(* IEC 61131-3 sources: elnaProjects/ElpcLogic/PomarKc7Changed/build_USO_ecl (part 2) *)

  ai.Tstali_statora_kanal_1.inCommand_ARM := UINT_TO_WORD(AI_Tstali_statora_kanal_1_command);
  ai.Tstali_statora_kanal_1.dHL := AI_Tstali_statora_kanal_1_newHL;
  ai.Tstali_statora_kanal_1.dLL := AI_Tstali_statora_kanal_1_newLL;
  ai.Tstali_statora_kanal_1.dHW := AI_Tstali_statora_kanal_1_newHW;

  ai.Tstali_statora_kanal_2.inCommand_ARM := UINT_TO_WORD(AI_Tstali_statora_kanal_2_command);
  ai.Tstali_statora_kanal_2.dHL := AI_Tstali_statora_kanal_2_newHL;
  ai.Tstali_statora_kanal_2.dLL := AI_Tstali_statora_kanal_2_newLL;
  ai.Tstali_statora_kanal_2.dHW := AI_Tstali_statora_kanal_2_newHW;

  ai.Tstali_statora_kanal_3.inCommand_ARM := UINT_TO_WORD(AI_Tstali_statora_kanal_3_command);
  ai.Tstali_statora_kanal_3.dHL := AI_Tstali_statora_kanal_3_newHL;
  ai.Tstali_statora_kanal_3.dLL := AI_Tstali_statora_kanal_3_newLL;
  ai.Tstali_statora_kanal_3.dHW := AI_Tstali_statora_kanal_3_newHW;

  ai.Tmedi_statora_kanal_1.inCommand_ARM := UINT_TO_WORD(AI_Tmedi_statora_kanal_1_command);
  ai.Tmedi_statora_kanal_1.dHL := AI_Tmedi_statora_kanal_1_newHL;
  ai.Tmedi_statora_kanal_1.dLL := AI_Tmedi_statora_kanal_1_newLL;
  ai.Tmedi_statora_kanal_1.dHW := AI_Tmedi_statora_kanal_1_newHW;

  ai.Tmedi_statora_kanal_2.inCommand_ARM := UINT_TO_WORD(AI_Tmedi_statora_kanal_2_command);
  ai.Tmedi_statora_kanal_2.dHL := AI_Tmedi_statora_kanal_2_newHL;
  ai.Tmedi_statora_kanal_2.dLL := AI_Tmedi_statora_kanal_2_newLL;
  ai.Tmedi_statora_kanal_2.dHW := AI_Tmedi_statora_kanal_2_newHW;

  ai.Tmedi_statora_kanal_3.inCommand_ARM := UINT_TO_WORD(AI_Tmedi_statora_kanal_3_command);
  ai.Tmedi_statora_kanal_3.dHL := AI_Tmedi_statora_kanal_3_newHL;
  ai.Tmedi_statora_kanal_3.dLL := AI_Tmedi_statora_kanal_3_newLL;
  ai.Tmedi_statora_kanal_3.dHW := AI_Tmedi_statora_kanal_3_newHW;

  ai.Toporno_podshipnika_EDT_1.inCommand_ARM := UINT_TO_WORD(AI_Toporno_podshipnika_EDT_1_command);
  ai.Toporno_podshipnika_EDT_1.dHL := AI_Toporno_podshipnika_EDT_1_newHL;
  ai.Toporno_podshipnika_EDT_1.dLL := AI_Toporno_podshipnika_EDT_1_newLL;
  ai.Toporno_podshipnika_EDT_1.dHW := AI_Toporno_podshipnika_EDT_1_newHW;
  ai.Toporno_podshipnika_EDT_1.dHA := AI_Toporno_podshipnika_EDT_1_newHA;

  ai.Toy_podshipnika_EDT_2.inCommand_ARM := UINT_TO_WORD(AI_Toy_podshipnika_EDT_2_command);
  ai.Toy_podshipnika_EDT_2.dHL := AI_Toy_podshipnika_EDT_2_newHL;
  ai.Toy_podshipnika_EDT_2.dLL := AI_Toy_podshipnika_EDT_2_newLL;
  ai.Toy_podshipnika_EDT_2.dHW := AI_Toy_podshipnika_EDT_2_newHW;
  ai.Toy_podshipnika_EDT_2.dHA := AI_Toy_podshipnika_EDT_2_newHA;

  ai.Toy_podshipnika_kol_EDT_3.inCommand_ARM := UINT_TO_WORD(AI_Toy_podshipnika_kol_EDT_3_command);
  ai.Toy_podshipnika_kol_EDT_3.dHL := AI_Toy_podshipnika_kol_EDT_3_newHL;
  ai.Toy_podshipnika_kol_EDT_3.dLL := AI_Toy_podshipnika_kol_EDT_3_newLL;
  ai.Toy_podshipnika_kol_EDT_3.dHW := AI_Toy_podshipnika_kol_EDT_3_newHW;
  ai.Toy_podshipnika_kol_EDT_3.dHA := AI_Toy_podshipnika_kol_EDT_3_newHA;

  ai.Toy_podshipnika_kol_EDT_4.inCommand_ARM := UINT_TO_WORD(AI_Toy_podshipnika_kol_EDT_4_command);
  ai.Toy_podshipnika_kol_EDT_4.dHL := AI_Toy_podshipnika_kol_EDT_4_newHL;
  ai.Toy_podshipnika_kol_EDT_4.dLL := AI_Toy_podshipnika_kol_EDT_4_newLL;
  ai.Toy_podshipnika_kol_EDT_4.dHW := AI_Toy_podshipnika_kol_EDT_4_newHW;
  ai.Toy_podshipnika_kol_EDT_4.dHA := AI_Toy_podshipnika_kol_EDT_4_newHA;

  ai.Toy_podshipnika_shest_red_EDT_5.inCommand_ARM := UINT_TO_WORD(AI_Toy_podshipnika_shest_red_EDT_5_command);
  ai.Toy_podshipnika_shest_red_EDT_5.dHL := AI_Toy_podshipnika_shest_red_EDT_5_newHL;
  ai.Toy_podshipnika_shest_red_EDT_5.dLL := AI_Toy_podshipnika_shest_red_EDT_5_newLL;
  ai.Toy_podshipnika_shest_red_EDT_5.dHW := AI_Toy_podshipnika_shest_red_EDT_5_newHW;
  ai.Toy_podshipnika_shest_red_EDT_5.dHA := AI_Toy_podshipnika_shest_red_EDT_5_newHA;

  ai.Ty_podshipnika_red_EDT_6.inCommand_ARM := UINT_TO_WORD(AI_Ty_podshipnika_red_EDT_6_command);
  ai.Ty_podshipnika_red_EDT_6.dHL := AI_Ty_podshipnika_red_EDT_6_newHL;
  ai.Ty_podshipnika_red_EDT_6.dLL := AI_Ty_podshipnika_red_EDT_6_newLL;
  ai.Ty_podshipnika_red_EDT_6.dHW := AI_Ty_podshipnika_red_EDT_6_newHW;
  ai.Ty_podshipnika_red_EDT_6.dHA := AI_Ty_podshipnika_red_EDT_6_newHA;

  ai.Ty_podshipnika_nagnet_EDT_7_1.inCommand_ARM := UINT_TO_WORD(AI_Ty_podshipnika_nagnet_EDT_7_1_command);
  ai.Ty_podshipnika_nagnet_EDT_7_1.dHL := AI_Ty_podshipnika_nagnet_EDT_7_1_newHL;
  ai.Ty_podshipnika_nagnet_EDT_7_1.dLL := AI_Ty_podshipnika_nagnet_EDT_7_1_newLL;
  ai.Ty_podshipnika_nagnet_EDT_7_1.dHW := AI_Ty_podshipnika_nagnet_EDT_7_1_newHW;
  ai.Ty_podshipnika_nagnet_EDT_7_1.dHA := AI_Ty_podshipnika_nagnet_EDT_7_1_newHA;

  ai.Ty_podshipnika_nagnet_EDT_7_2.inCommand_ARM := UINT_TO_WORD(AI_Ty_podshipnika_nagnet_EDT_7_2_command);
  ai.Ty_podshipnika_nagnet_EDT_7_2.dHL := AI_Ty_podshipnika_nagnet_EDT_7_2_newHL;
  ai.Ty_podshipnika_nagnet_EDT_7_2.dLL := AI_Ty_podshipnika_nagnet_EDT_7_2_newLL;
  ai.Ty_podshipnika_nagnet_EDT_7_2.dHW := AI_Ty_podshipnika_nagnet_EDT_7_2_newHW;
  ai.Ty_podshipnika_nagnet_EDT_7_2.dHA := AI_Ty_podshipnika_nagnet_EDT_7_2_newHA;

  ai.Toy_podshipnika_svobod_konca_EDT_8_1.inCommand_ARM := UINT_TO_WORD(AI_Toy_podshipnika_svobod_konca_EDT_8_1_command);
  ai.Toy_podshipnika_svobod_konca_EDT_8_1.dHL := AI_Toy_podshipnika_svobod_konca_EDT_8_1_newHL;
  ai.Toy_podshipnika_svobod_konca_EDT_8_1.dLL := AI_Toy_podshipnika_svobod_konca_EDT_8_1_newLL;
  ai.Toy_podshipnika_svobod_konca_EDT_8_1.dHW := AI_Toy_podshipnika_svobod_konca_EDT_8_1_newHW;
  ai.Toy_podshipnika_svobod_konca_EDT_8_1.dHA := AI_Toy_podshipnika_svobod_konca_EDT_8_1_newHA;

  ai.Toy_podshipnika_svobod_konca_EDT_8_2.inCommand_ARM := UINT_TO_WORD(AI_Toy_podshipnika_svobod_konca_EDT_8_2_command);
  ai.Toy_podshipnika_svobod_konca_EDT_8_2.dHL := AI_Toy_podshipnika_svobod_konca_EDT_8_2_newHL;
  ai.Toy_podshipnika_svobod_konca_EDT_8_2.dLL := AI_Toy_podshipnika_svobod_konca_EDT_8_2_newLL;
  ai.Toy_podshipnika_svobod_konca_EDT_8_2.dHW := AI_Toy_podshipnika_svobod_konca_EDT_8_2_newHW;
  ai.Toy_podshipnika_svobod_konca_EDT_8_2.dHA := AI_Toy_podshipnika_svobod_konca_EDT_8_2_newHA;

  ai.Toy_podshipnika_rab_kol_EDT_9_1.inCommand_ARM := UINT_TO_WORD(AI_Toy_podshipnika_rab_kol_EDT_9_1_command);
  ai.Toy_podshipnika_rab_kol_EDT_9_1.dHL := AI_Toy_podshipnika_rab_kol_EDT_9_1_newHL;
  ai.Toy_podshipnika_rab_kol_EDT_9_1.dLL := AI_Toy_podshipnika_rab_kol_EDT_9_1_newLL;
  ai.Toy_podshipnika_rab_kol_EDT_9_1.dHW := AI_Toy_podshipnika_rab_kol_EDT_9_1_newHW;
  ai.Toy_podshipnika_rab_kol_EDT_9_1.dHA := AI_Toy_podshipnika_rab_kol_EDT_9_1_newHA;

  ai.Toy_podshipnika_rab_kol_EDT_9_2.inCommand_ARM := UINT_TO_WORD(AI_Toy_podshipnika_rab_kol_EDT_9_2_command);
  ai.Toy_podshipnika_rab_kol_EDT_9_2.dHL := AI_Toy_podshipnika_rab_kol_EDT_9_2_newHL;
  ai.Toy_podshipnika_rab_kol_EDT_9_2.dLL := AI_Toy_podshipnika_rab_kol_EDT_9_2_newLL;
  ai.Toy_podshipnika_rab_kol_EDT_9_2.dHW := AI_Toy_podshipnika_rab_kol_EDT_9_2_newHW;
  ai.Toy_podshipnika_rab_kol_EDT_9_2.dHA := AI_Toy_podshipnika_rab_kol_EDT_9_2_newHA;

  ai.Toy_podshipnika_nerab_kol_EDT_10_1.inCommand_ARM := UINT_TO_WORD(AI_Toy_podshipnika_nerab_kol_EDT_10_1_command);
  ai.Toy_podshipnika_nerab_kol_EDT_10_1.dHL := AI_Toy_podshipnika_nerab_kol_EDT_10_1_newHL;
  ai.Toy_podshipnika_nerab_kol_EDT_10_1.dLL := AI_Toy_podshipnika_nerab_kol_EDT_10_1_newLL;
  ai.Toy_podshipnika_nerab_kol_EDT_10_1.dHW := AI_Toy_podshipnika_nerab_kol_EDT_10_1_newHW;
  ai.Toy_podshipnika_nerab_kol_EDT_10_1.dHA := AI_Toy_podshipnika_nerab_kol_EDT_10_1_newHA;

  ai.Toy_podshipnika_nerab_kol_EDT_10_2.inCommand_ARM := UINT_TO_WORD(AI_Toy_podshipnika_nerab_kol_EDT_10_2_command);
  ai.Toy_podshipnika_nerab_kol_EDT_10_2.dHL := AI_Toy_podshipnika_nerab_kol_EDT_10_2_newHL;
  ai.Toy_podshipnika_nerab_kol_EDT_10_2.dLL := AI_Toy_podshipnika_nerab_kol_EDT_10_2_newLL;
  ai.Toy_podshipnika_nerab_kol_EDT_10_2.dHW := AI_Toy_podshipnika_nerab_kol_EDT_10_2_newHW;
  ai.Toy_podshipnika_nerab_kol_EDT_10_2.dHA := AI_Toy_podshipnika_nerab_kol_EDT_10_2_newHA;

  ai.Tholodnogo_vozduha_ED_kanal_1.inCommand_ARM := UINT_TO_WORD(AI_Tholodnogo_vozduha_ED_kanal_1_command);
  ai.Tholodnogo_vozduha_ED_kanal_1.dHL := AI_Tholodnogo_vozduha_ED_kanal_1_newHL;
  ai.Tholodnogo_vozduha_ED_kanal_1.dLL := AI_Tholodnogo_vozduha_ED_kanal_1_newLL;
  ai.Tholodnogo_vozduha_ED_kanal_1.dHW := AI_Tholodnogo_vozduha_ED_kanal_1_newHW;

  ai.Tholodnogo_vozduha_ED_kanal_2.inCommand_ARM := UINT_TO_WORD(AI_Tholodnogo_vozduha_ED_kanal_2_command);
  ai.Tholodnogo_vozduha_ED_kanal_2.dHL := AI_Tholodnogo_vozduha_ED_kanal_2_newHL;
  ai.Tholodnogo_vozduha_ED_kanal_2.dLL := AI_Tholodnogo_vozduha_ED_kanal_2_newLL;
  ai.Tholodnogo_vozduha_ED_kanal_2.dHW := AI_Tholodnogo_vozduha_ED_kanal_2_newHW;

  ai.Tgorjachego_vozduha_ED_kanal_1.inCommand_ARM := UINT_TO_WORD(AI_Tgorjachego_vozduha_ED_kanal_1_command);
  ai.Tgorjachego_vozduha_ED_kanal_1.dHL := AI_Tgorjachego_vozduha_ED_kanal_1_newHL;
  ai.Tgorjachego_vozduha_ED_kanal_1.dLL := AI_Tgorjachego_vozduha_ED_kanal_1_newLL;
  ai.Tgorjachego_vozduha_ED_kanal_1.dHW := AI_Tgorjachego_vozduha_ED_kanal_1_newHW;

  ai.Tgorjachego_vozduha_ED_kanal_2.inCommand_ARM := UINT_TO_WORD(AI_Tgorjachego_vozduha_ED_kanal_2_command);
  ai.Tgorjachego_vozduha_ED_kanal_2.dHL := AI_Tgorjachego_vozduha_ED_kanal_2_newHL;
  ai.Tgorjachego_vozduha_ED_kanal_2.dLL := AI_Tgorjachego_vozduha_ED_kanal_2_newLL;
  ai.Tgorjachego_vozduha_ED_kanal_2.dHW := AI_Tgorjachego_vozduha_ED_kanal_2_newHW;

  ai.Tnarujnogo_vozduha.inCommand_ARM := UINT_TO_WORD(AI_Tnarujnogo_vozduha_command);
  ai.Tnarujnogo_vozduha.dHL := AI_Tnarujnogo_vozduha_newHL;
  ai.Tnarujnogo_vozduha.dLL := AI_Tnarujnogo_vozduha_newLL;
  ai.Tnarujnogo_vozduha.dHW := AI_Tnarujnogo_vozduha_newHW;

  ai.Tgaza_na_vhode_H.inCommand_ARM := UINT_TO_WORD(AI_Tgaza_na_vhode_H_command);
  ai.Tgaza_na_vhode_H.dHL := AI_Tgaza_na_vhode_H_newHL;
  ai.Tgaza_na_vhode_H.dLL := AI_Tgaza_na_vhode_H_newLL;
  ai.Tgaza_na_vhode_H.dHW := AI_Tgaza_na_vhode_H_newHW;

  ai.Tgaza_na_vyhode_H.inCommand_ARM := UINT_TO_WORD(AI_Tgaza_na_vyhode_H_command);
  ai.Tgaza_na_vyhode_H.dHL := AI_Tgaza_na_vyhode_H_newHL;
  ai.Tgaza_na_vyhode_H.dLL := AI_Tgaza_na_vyhode_H_newLL;
  ai.Tgaza_na_vyhode_H.dHW := AI_Tgaza_na_vyhode_H_newHW;
  ai.Tgaza_na_vyhode_H.dHA := AI_Tgaza_na_vyhode_H_newHA;

  ai.Tmasla_do_AVOM.inCommand_ARM := UINT_TO_WORD(AI_Tmasla_do_AVOM_command);
  ai.Tmasla_do_AVOM.dHL := AI_Tmasla_do_AVOM_newHL;
  ai.Tmasla_do_AVOM.dLL := AI_Tmasla_do_AVOM_newLL;
  ai.Tmasla_do_AVOM.dHW := AI_Tmasla_do_AVOM_newHW;

  ai.Tmasla_posle_AVOM.inCommand_ARM := UINT_TO_WORD(AI_Tmasla_posle_AVOM_command);
  ai.Tmasla_posle_AVOM.dHL := AI_Tmasla_posle_AVOM_newHL;
  ai.Tmasla_posle_AVOM.dLL := AI_Tmasla_posle_AVOM_newLL;
  ai.Tmasla_posle_AVOM.dHW := AI_Tmasla_posle_AVOM_newHW;

  ai.Tmasla_MB.inCommand_ARM := UINT_TO_WORD(AI_Tmasla_MB_command);
  ai.Tmasla_MB.dHL := AI_Tmasla_MB_newHL;
  ai.Tmasla_MB.dLL := AI_Tmasla_MB_newLL;
  ai.Tmasla_MB.dHW := AI_Tmasla_MB_newHW;

  ai.Tmasla_MB_TEN.inCommand_ARM := UINT_TO_WORD(AI_Tmasla_MB_TEN_command);
  ai.Tmasla_MB_TEN.dHL := AI_Tmasla_MB_TEN_newHL;
  ai.Tmasla_MB_TEN.dLL := AI_Tmasla_MB_TEN_newLL;
  ai.Tmasla_MB_TEN.dHW := AI_Tmasla_MB_TEN_newHW;

  ai.Tshu.inCommand_ARM := UINT_TO_WORD(AI_Tshu_command);
  ai.Tshu.dHL := AI_Tshu_newHL;
  ai.Tshu.dLL := AI_Tshu_newLL;

  ai.Pmaslo_sm_nizkoe.inCommand_ARM := UINT_TO_WORD(AI_Pmaslo_sm_nizkoe_command);
  ai.Pmaslo_sm_nizkoe.dHL := AI_Pmaslo_sm_nizkoe_newHL;
  ai.Pmaslo_sm_nizkoe.dLL := AI_Pmaslo_sm_nizkoe_newLL;
  ai.Pmaslo_sm_nizkoe.dLW := AI_Pmaslo_sm_nizkoe_newLW;
  ai.Pmaslo_sm_nizkoe.dLA := AI_Pmaslo_sm_nizkoe_newLA;

  ai.Pmaslo_sm_vysokoe.inCommand_ARM := UINT_TO_WORD(AI_Pmaslo_sm_vysokoe_command);
  ai.Pmaslo_sm_vysokoe.dHL := AI_Pmaslo_sm_vysokoe_newHL;
  ai.Pmaslo_sm_vysokoe.dLL := AI_Pmaslo_sm_vysokoe_newLL;
  ai.Pmaslo_sm_vysokoe.dLW := AI_Pmaslo_sm_vysokoe_newLW;
  ai.Pmaslo_sm_vysokoe.dLA := AI_Pmaslo_sm_vysokoe_newLA;

  ai.Pmasla_posle_GNS.inCommand_ARM := UINT_TO_WORD(AI_Pmasla_posle_GNS_command);
  ai.Pmasla_posle_GNS.dHL := AI_Pmasla_posle_GNS_newHL;
  ai.Pmasla_posle_GNS.dLL := AI_Pmasla_posle_GNS_newLL;
  ai.Pmasla_posle_GNS.dHW := AI_Pmasla_posle_GNS_newHW;
  ai.Pmasla_posle_GNS.dLW := AI_Pmasla_posle_GNS_newLW;

  ai.Pmasla_posle_NU.inCommand_ARM := UINT_TO_WORD(AI_Pmasla_posle_NU_command);
  ai.Pmasla_posle_NU.dHL := AI_Pmasla_posle_NU_newHL;
  ai.Pmasla_posle_NU.dLL := AI_Pmasla_posle_NU_newLL;
  ai.Pmasla_posle_NU.dLW := AI_Pmasla_posle_NU_newLW;

  ai.Pgaza_na_vhode_nagnetatelia.inCommand_ARM := UINT_TO_WORD(AI_Pgaza_na_vhode_nagnetatelia_command);
  ai.Pgaza_na_vhode_nagnetatelia.dHL := AI_Pgaza_na_vhode_nagnetatelia_newHL;
  ai.Pgaza_na_vhode_nagnetatelia.dLL := AI_Pgaza_na_vhode_nagnetatelia_newLL;
  ai.Pgaza_na_vhode_nagnetatelia.dLW := AI_Pgaza_na_vhode_nagnetatelia_newLW;

  ai.Pgaza_na_vyhode_nagnetatelia.inCommand_ARM := UINT_TO_WORD(AI_Pgaza_na_vyhode_nagnetatelia_command);
  ai.Pgaza_na_vyhode_nagnetatelia.dHL := AI_Pgaza_na_vyhode_nagnetatelia_newHL;
  ai.Pgaza_na_vyhode_nagnetatelia.dLL := AI_Pgaza_na_vyhode_nagnetatelia_newLL;
  ai.Pgaza_na_vyhode_nagnetatelia.dLW := AI_Pgaza_na_vyhode_nagnetatelia_newLW;
  ai.Pgaza_na_vyhode_nagnetatelia.dHA := AI_Pgaza_na_vyhode_nagnetatelia_newHA;

  ai.Pimpuls_gaz.inCommand_ARM := UINT_TO_WORD(AI_Pimpuls_gaz_command);
  ai.Pimpuls_gaz.dHL := AI_Pimpuls_gaz_newHL;
  ai.Pimpuls_gaz.dLL := AI_Pimpuls_gaz_newLL;
  ai.Pimpuls_gaz.dLW := AI_Pimpuls_gaz_newLW;

  ai.dPgaza_na_maslo_filtre.inCommand_ARM := UINT_TO_WORD(AI_dPgaza_na_maslo_filtre_command);
  ai.dPgaza_na_maslo_filtre.dHL := AI_dPgaza_na_maslo_filtre_newHL;
  ai.dPgaza_na_maslo_filtre.dLL := AI_dPgaza_na_maslo_filtre_newLL;
  ai.dPgaza_na_maslo_filtre.dHW := AI_dPgaza_na_maslo_filtre_newHW;

  ai.dPgaza_na_konfuzore.inCommand_ARM := UINT_TO_WORD(AI_dPgaza_na_konfuzore_command);
  ai.dPgaza_na_konfuzore.dHL := AI_dPgaza_na_konfuzore_newHL;
  ai.dPgaza_na_konfuzore.dLL := AI_dPgaza_na_konfuzore_newLL;
  ai.dPgaza_na_konfuzore.dLW := AI_dPgaza_na_konfuzore_newLW;

  ai.dPmaslo_gaz.inCommand_ARM := UINT_TO_WORD(AI_dPmaslo_gaz_command);
  ai.dPmaslo_gaz.dHL := AI_dPmaslo_gaz_newHL;
  ai.dPmaslo_gaz.dLL := AI_dPmaslo_gaz_newLL;
  ai.dPmaslo_gaz.dLW := AI_dPmaslo_gaz_newLW;
  ai.dPmaslo_gaz.dLA := AI_dPmaslo_gaz_newLA;

  ai.Os_sdvig_nagnetatelja_plus.inCommand_ARM := UINT_TO_WORD(AI_Os_sdvig_nagnetatelja_plus_command);
  ai.Os_sdvig_nagnetatelja_plus.dHL := AI_Os_sdvig_nagnetatelja_plus_newHL;
  ai.Os_sdvig_nagnetatelja_plus.dLL := AI_Os_sdvig_nagnetatelja_plus_newLL;
  ai.Os_sdvig_nagnetatelja_plus.dHW := AI_Os_sdvig_nagnetatelja_plus_newHW;
  ai.Os_sdvig_nagnetatelja_plus.dHA := AI_Os_sdvig_nagnetatelja_plus_newHA;

  ai.Os_sdvig_nagnetatelja_minus.inCommand_ARM := UINT_TO_WORD(AI_Os_sdvig_nagnetatelja_minus_command);
  ai.Os_sdvig_nagnetatelja_minus.dHL := AI_Os_sdvig_nagnetatelja_minus_newHL;
  ai.Os_sdvig_nagnetatelja_minus.dLL := AI_Os_sdvig_nagnetatelja_minus_newLL;
  ai.Os_sdvig_nagnetatelja_minus.dLW := AI_Os_sdvig_nagnetatelja_minus_newLW;
  ai.Os_sdvig_nagnetatelja_minus.dLA := AI_Os_sdvig_nagnetatelja_minus_newLA;

  ai.Yroven_masla_MB.inCommand_ARM := UINT_TO_WORD(AI_Yroven_masla_MB_command);
  ai.Yroven_masla_MB.dHL := AI_Yroven_masla_MB_newHL;
  ai.Yroven_masla_MB.dLL := AI_Yroven_masla_MB_newLL;
  ai.Yroven_masla_MB.dLW := AI_Yroven_masla_MB_newLW;

  ai.Kontrol_per_220V.inCommand_ARM := UINT_TO_WORD(AI_Kontrol_per_220V_command);
  ai.Kontrol_per_220V.dHL := AI_Kontrol_per_220V_newHL;
  ai.Kontrol_per_220V.dLL := AI_Kontrol_per_220V_newLL;
  ai.Kontrol_per_220V.dHW := AI_Kontrol_per_220V_newHW;
  ai.Kontrol_per_220V.dLW := AI_Kontrol_per_220V_newLW;

  ai.Kontrol_post_220V.inCommand_ARM := UINT_TO_WORD(AI_Kontrol_post_220V_command);
  ai.Kontrol_post_220V.dHL := AI_Kontrol_post_220V_newHL;
  ai.Kontrol_post_220V.dLL := AI_Kontrol_post_220V_newLL;
  ai.Kontrol_post_220V.dHW := AI_Kontrol_post_220V_newHW;
  ai.Kontrol_post_220V.dLW := AI_Kontrol_post_220V_newLW;

  ai.Tok_statora.inCommand_ARM := UINT_TO_WORD(AI_Tok_statora_command);
  ai.Tok_statora.dHL := AI_Tok_statora_newHL;
  ai.Tok_statora.dLL := AI_Tok_statora_newLL;
  ai.Tok_statora.dLW := AI_Tok_statora_newLW;

  ai.Vibro_skorost_OPED_T1.inCommand_ARM := UINT_TO_WORD(AI_Vibro_skorost_OPED_T1_command);
  ai.Vibro_skorost_OPED_T1.dHL := AI_Vibro_skorost_OPED_T1_newHL;
  ai.Vibro_skorost_OPED_T1.dLL := AI_Vibro_skorost_OPED_T1_newLL;
  ai.Vibro_skorost_OPED_T1.dHW := AI_Vibro_skorost_OPED_T1_newHW;
  ai.Vibro_skorost_OPED_T1.dHA := AI_Vibro_skorost_OPED_T1_newHA;

  ai.Vibro_skorost_OYPED_T2.inCommand_ARM := UINT_TO_WORD(AI_Vibro_skorost_OYPED_T2_command);
  ai.Vibro_skorost_OYPED_T2.dHL := AI_Vibro_skorost_OYPED_T2_newHL;
  ai.Vibro_skorost_OYPED_T2.dLL := AI_Vibro_skorost_OYPED_T2_newLL;
  ai.Vibro_skorost_OYPED_T2.dHW := AI_Vibro_skorost_OYPED_T2_newHW;
  ai.Vibro_skorost_OYPED_T2.dHA := AI_Vibro_skorost_OYPED_T2_newHA;

  ai.Vibro_skorost_OYP_kolesa_ED_T3.inCommand_ARM := UINT_TO_WORD(AI_Vibro_skorost_OYP_kolesa_ED_T3_command);
  ai.Vibro_skorost_OYP_kolesa_ED_T3.dHL := AI_Vibro_skorost_OYP_kolesa_ED_T3_newHL;
  ai.Vibro_skorost_OYP_kolesa_ED_T3.dLL := AI_Vibro_skorost_OYP_kolesa_ED_T3_newLL;
  ai.Vibro_skorost_OYP_kolesa_ED_T3.dHW := AI_Vibro_skorost_OYP_kolesa_ED_T3_newHW;
  ai.Vibro_skorost_OYP_kolesa_ED_T3.dHA := AI_Vibro_skorost_OYP_kolesa_ED_T3_newHA;

  ai.Vibro_skorost_OP_kolesa_RH_T4.inCommand_ARM := UINT_TO_WORD(AI_Vibro_skorost_OP_kolesa_RH_T4_command);
  ai.Vibro_skorost_OP_kolesa_RH_T4.dHL := AI_Vibro_skorost_OP_kolesa_RH_T4_newHL;
  ai.Vibro_skorost_OP_kolesa_RH_T4.dLL := AI_Vibro_skorost_OP_kolesa_RH_T4_newLL;
  ai.Vibro_skorost_OP_kolesa_RH_T4.dHW := AI_Vibro_skorost_OP_kolesa_RH_T4_newHW;
  ai.Vibro_skorost_OP_kolesa_RH_T4.dHA := AI_Vibro_skorost_OP_kolesa_RH_T4_newHA;

  ai.Vibro_skorost_OP_shesterni_RED_T5.inCommand_ARM := UINT_TO_WORD(AI_Vibro_skorost_OP_shesterni_RED_T5_command);
  ai.Vibro_skorost_OP_shesterni_RED_T5.dHL := AI_Vibro_skorost_OP_shesterni_RED_T5_newHL;
  ai.Vibro_skorost_OP_shesterni_RED_T5.dLL := AI_Vibro_skorost_OP_shesterni_RED_T5_newLL;
  ai.Vibro_skorost_OP_shesterni_RED_T5.dHW := AI_Vibro_skorost_OP_shesterni_RED_T5_newHW;
  ai.Vibro_skorost_OP_shesterni_RED_T5.dHA := AI_Vibro_skorost_OP_shesterni_RED_T5_newHA;

  ai.Vibro_skorost_OP_shesterni_RED_T6.inCommand_ARM := UINT_TO_WORD(AI_Vibro_skorost_OP_shesterni_RED_T6_command);
  ai.Vibro_skorost_OP_shesterni_RED_T6.dHL := AI_Vibro_skorost_OP_shesterni_RED_T6_newHL;
  ai.Vibro_skorost_OP_shesterni_RED_T6.dLL := AI_Vibro_skorost_OP_shesterni_RED_T6_newLL;
  ai.Vibro_skorost_OP_shesterni_RED_T6.dHW := AI_Vibro_skorost_OP_shesterni_RED_T6_newHW;
  ai.Vibro_skorost_OP_shesterni_RED_T6.dHA := AI_Vibro_skorost_OP_shesterni_RED_T6_newHA;
END_FUNCTION_BLOCK

FUNCTION_BLOCK fb_ph_Timer
  VAR_INPUT
    delay : TIME;
    PhaseNumber : UINT;
  END_VAR
  VAR_IN_OUT
    StrPh : struct_PhaseAlgoritm;
  END_VAR
  VAR
    CommandFault_Trig : R_TRIG;
    reset_Trig : R_TRIG;
  END_VAR
  VAR_IN_OUT
    timer : UINT;
  END_VAR
  VAR
    _timer : TON;
    _statusDualInput : TYPE_statusDualInput;
  END_VAR

  IF StrPh.run AND NOT StrPh.start THEN
  	StrPh.start := TRUE;
  	StrPh.top := FALSE;
  	StrPh.error := FALSE;
            StrPh.run:=FALSE;

  END_IF;

  _timer(IN:=StrPh.start, PT:=delay);

  timer:=TIME_TO_UINT(delay -_timer.ET);

  IF StrPh.start AND NOT StrPh.top THEN
  StrPh.top:=_timer.Q;
  END_IF;

  reset_Trig(CLK := StrPh.reset);
  IF reset_Trig.Q THEN
  	StrPh.start := FALSE;
  	StrPh.error := FALSE;
  	StrPh.top := FALSE;
            StrPh.run:=FALSE;
            (*timer:=TIME_TO_UINT(delay -_timer.ET);*)
            StrPh.reset:=FALSE;
  END_IF;

  StrPh.startStatus := SHL(BOOL_TO_DWORD(StrPh.start), PhaseNumber);
  StrPh.errorStatus := SHL(BOOL_TO_DWORD(StrPh.error), PhaseNumber);
  StrPh.topStatus := SHL(BOOL_TO_DWORD(StrPh.top), PhaseNumber);
END_FUNCTION_BLOCK

FUNCTION_BLOCK fb_ph_Kran
  VAR_IN_OUT
    im : struct_Kran;
    StrPh : struct_PhaseAlgoritm;
  END_VAR
  VAR_INPUT
    act : TYPE_DualStateImAction;
    PhaseNumber : UINT;
  END_VAR
  VAR
    CommandFault_Trig : R_TRIG;
    reset_Trig : R_TRIG;
    _statusDualInput : TYPE_statusDualInput;
  END_VAR

  IF StrPh.run AND NOT StrPh.start THEN
  	StrPh.start := TRUE;
  	StrPh.top := FALSE;
  	StrPh.error := FALSE;
            StrPh.run:=FALSE;

  	CASE act OF
  		(*DualStateImAction.on*)   _on: im.inOpcCommandsDisabled:=TRUE;
                                                      im.inCommand_Alg := 1; (*cmd_open*)
  		(*DualStateImAction.off*) _off: im.inOpcCommandsDisabled:=TRUE;
                                                      im.inCommand_Alg := 2; (*cmd_close*)
  	END_CASE;
  END_IF;

  IF StrPh.start AND NOT StrPh.top THEN
                      CommandFault_Trig(CLK := im.CommandFault);
                      IF CommandFault_Trig.Q THEN
  	          StrPh.error := TRUE;
                      END_IF;

  		CASE act OF
  		(*_DualStateImAction.on*)    _on: StrPh.top := im.onStatus = _statusDualInput.STATUS_ON;
  		(*_DualStateImAction.off*)  _off: StrPh.top := im.onStatus = _statusDualInput.STATUS_OFF;
  		END_CASE;

  END_IF;

  IF StrPh.top THEN
  StrPh.error := FALSE;
  END_IF;

  reset_Trig(CLK := StrPh.reset);
  IF reset_Trig.Q THEN
  	StrPh.start := FALSE;
  	StrPh.error := FALSE;
  	StrPh.top := FALSE;
            StrPh.run:=FALSE;
            StrPh.reset:=FALSE;
  END_IF;

  StrPh.startStatus := SHL(BOOL_TO_DWORD(StrPh.start), PhaseNumber);
  StrPh.errorStatus := SHL(BOOL_TO_DWORD(StrPh.error), PhaseNumber);
  StrPh.topStatus := SHL(BOOL_TO_DWORD(StrPh.top), PhaseNumber);
END_FUNCTION_BLOCK

FUNCTION_BLOCK fb_ph_Switch
  VAR_IN_OUT
    im : struct_Switch;
  END_VAR
  VAR_INPUT
    act : TYPE_DualStateImAction;
    PhaseNumber : UINT;
  END_VAR
  VAR_IN_OUT
    StrPh : struct_PhaseAlgoritm;
  END_VAR
  VAR
    CommandFault_Trig : R_TRIG;
    reset_Trig : R_TRIG;
    _statusDualInput : TYPE_statusDualInput;
  END_VAR

  IF StrPh.run AND NOT StrPh.start THEN
  	StrPh.start := TRUE;
  	StrPh.top := FALSE;
  	StrPh.error := FALSE;
            StrPh.run:=FALSE;

  	CASE act OF
  		(*DualStateImAction.on*)   _on :im.inOpcCommandsDisabled:=TRUE;
                                                      im.inCommand_Alg := 1; (*cmd_open*)
  		(*DualStateImAction.off*) _off :im.inOpcCommandsDisabled:=TRUE;
                                                      im.inCommand_Alg := 2; (*cmd_close*)
  	END_CASE;
  END_IF;

  IF StrPh.start AND NOT StrPh.top THEN
                      CommandFault_Trig(CLK := im.CommandFault);
                      IF CommandFault_Trig.Q THEN
  	          StrPh.error := TRUE;
                      END_IF;

  		CASE act OF
  		(*_DualStateImAction.on*)    _on: StrPh.top := im.onStatus = _statusDualInput.STATUS_ON;
  		(*_DualStateImAction.off*)  _off: StrPh.top := im.onStatus = _statusDualInput.STATUS_OFF;
  		END_CASE;

  END_IF;

  IF StrPh.top THEN
  StrPh.error := FALSE;
  END_IF;

  reset_Trig(CLK := StrPh.reset);
  IF reset_Trig.Q THEN
  	StrPh.start := FALSE;
  	StrPh.error := FALSE;
  	StrPh.top := FALSE;
            StrPh.run:=FALSE;
            StrPh.reset:=FALSE;
  END_IF;

  StrPh.startStatus := SHL(BOOL_TO_DWORD(StrPh.start), PhaseNumber);
  StrPh.errorStatus := SHL(BOOL_TO_DWORD(StrPh.error), PhaseNumber);
  StrPh.topStatus := SHL(BOOL_TO_DWORD(StrPh.top), PhaseNumber);
END_FUNCTION_BLOCK

FUNCTION_BLOCK fb_ph_SectionSwitch
  VAR_IN_OUT
    im : struct_SectionSwitch;
  END_VAR
  VAR_INPUT
    act : TYPE_DualStateImAction;
    PhaseNumber : UINT;
  END_VAR
  VAR_IN_OUT
    StrPh : struct_PhaseAlgoritm;
  END_VAR
  VAR
    CommandFault_Trig : R_TRIG;
    reset_Trig : R_TRIG;
    _statusDualInput : TYPE_statusDualInput;
  END_VAR

  IF StrPh.run AND NOT StrPh.start THEN
  	StrPh.start := TRUE;
  	StrPh.top := FALSE;
  	StrPh.error := FALSE;
            StrPh.run:=FALSE;

  	CASE act OF
  		(*DualStateImAction.on*)   _on : im.inOpcCommandsDisabled:=TRUE;
                                                       im.inCommand_Alg := 1; (*cmd_open*)
  		(*DualStateImAction.off*) _off : im.inOpcCommandsDisabled:=TRUE;
                                                       im.inCommand_Alg := 2; (*cmd_close*)
  	END_CASE;
  END_IF;

  IF StrPh.start AND NOT StrPh.top THEN
                      CommandFault_Trig(CLK := im.CommandFault);
                      IF CommandFault_Trig.Q THEN
  	          StrPh.error := TRUE;
                      END_IF;

  		CASE act OF
  		(*_DualStateImAction.on*)    _on: StrPh.top := im.onStatus = _statusDualInput.STATUS_ON;
  		(*_DualStateImAction.off*)  _off: StrPh.top := im.onStatus = _statusDualInput.STATUS_OFF;
  		END_CASE;

  END_IF;

  IF StrPh.top THEN
  StrPh.error := FALSE;
  END_IF;

  reset_Trig(CLK := StrPh.reset);
  IF reset_Trig.Q THEN
  	StrPh.start := FALSE;
  	StrPh.error := FALSE;
  	StrPh.top := FALSE;
            StrPh.run:=FALSE;
            StrPh.reset:=FALSE;
  END_IF;

  StrPh.startStatus := SHL(BOOL_TO_DWORD(StrPh.start), PhaseNumber);
  StrPh.errorStatus := SHL(BOOL_TO_DWORD(StrPh.error), PhaseNumber);
  StrPh.topStatus := SHL(BOOL_TO_DWORD(StrPh.top), PhaseNumber);
END_FUNCTION_BLOCK

FUNCTION_BLOCK fb_ph_CustomPhase
  VAR_INPUT
    PhaseNumber : UINT;
  END_VAR
  VAR_IN_OUT
    StrPh : struct_PhaseAlgoritm;
  END_VAR
  VAR
    CommandFault_Trig : R_TRIG;
    reset_Trig : R_TRIG;
    _statusDualInput : TYPE_statusDualInput;
  END_VAR

  IF StrPh.run AND NOT StrPh.start THEN
  	StrPh.start := TRUE;
  	StrPh.top := FALSE;
  	StrPh.error := FALSE;
            StrPh.run:=FALSE;
  END_IF;

  IF StrPh.top THEN StrPh.error := FALSE; END_IF;

  reset_Trig(CLK := StrPh.reset);
  IF reset_Trig.Q THEN
  	StrPh.start := FALSE;
  	StrPh.error := FALSE;
  	StrPh.top := FALSE;
            StrPh.run:=FALSE;
            StrPh.reset:=FALSE;
  END_IF;

  StrPh.startStatus := SHL(BOOL_TO_DWORD(StrPh.start), PhaseNumber);
  StrPh.errorStatus := SHL(BOOL_TO_DWORD(StrPh.error), PhaseNumber);
  StrPh.topStatus := SHL(BOOL_TO_DWORD(StrPh.top), PhaseNumber);
END_FUNCTION_BLOCK

FUNCTION resetIfRunning : BOOL
  VAR_IN_OUT
    alg : struct_Alg;
  END_VAR
  VAR CONSTANT
    cmdReset : WORD          := 2;
  END_VAR

  IF alg.isRuning THEN
                      alg.inOpcCommandsDisabled:=TRUE;
  		alg.inCommand_Alg:=cmdReset;
  END_IF;
END_FUNCTION

FUNCTION runIfNotRunning : BOOL
  VAR_IN_OUT
    alg : struct_Alg;
  END_VAR
  VAR CONSTANT
    cmdRun : WORD          := 1;
  END_VAR

  IF NOT alg.isRuning THEN
                      alg.inOpcCommandsDisabled:=TRUE;
                      alg.inCanRun:=TRUE;
  		alg.inCommand_Alg:=cmdRun;
  END_IF;
END_FUNCTION

FUNCTION_BLOCK fb_ph_algoritm
  VAR_IN_OUT
    alg : struct_Alg;
  END_VAR
  VAR_INPUT
    act : TYPE_PhaseAlgoritmAction;
    PhaseNumber : UINT;
    waitCompletion : BOOL;
  END_VAR
  VAR_IN_OUT
    StrPh : struct_PhaseAlgoritm;
  END_VAR
  VAR
    CommandFault_Trig : R_TRIG;
    reset_Trig : R_TRIG;
    _statusDualInput : TYPE_statusDualInput;
  END_VAR

  IF StrPh.run AND NOT StrPh.start THEN
  	StrPh.start := TRUE;
  	StrPh.top := FALSE;
  	StrPh.error := FALSE;
            StrPh.run:=FALSE;

  	CASE act OF
  		(*PhaseAlgoritmAction.run*)    _run : runIfNotRunning(alg); (*cmd_run*)
  		(*PhaseAlgoritmAction.reset*)_reset : resetIfRunning(alg); (*cmd_reset*)
  	END_CASE;
  END_IF;

  IF StrPh.start AND NOT StrPh.top THEN
                      CommandFault_Trig(CLK := alg.hasError);
                      IF CommandFault_Trig.Q THEN
  	          StrPh.error := TRUE;
                      END_IF;

  		CASE act OF
  		(*PhaseAlgoritmAction.run*)    _run:
                                                          IF waitCompletion THEN
  		                                	StrPh.top:=alg.isEnded;
  		                                    ELSE
  			                              StrPh.top:=alg.isRuning;
  		                                    END_IF;

  		(*PhaseAlgoritmAction.reset*) _reset:   StrPh.top := NOT alg.isRuning;
  		END_CASE;

  END_IF;

  IF StrPh.top THEN
  StrPh.error := FALSE;
  END_IF;

  reset_Trig(CLK := StrPh.reset);
  IF reset_Trig.Q THEN
            IF waitCompletion THEN
            resetIfRunning(alg);
            END_IF;
  	StrPh.start := FALSE;
  	StrPh.error := FALSE;
  	StrPh.top := FALSE;
            StrPh.run:=FALSE;
            StrPh.reset:=FALSE;
  END_IF;

  StrPh.startStatus := SHL(BOOL_TO_DWORD(StrPh.start), PhaseNumber);
  StrPh.errorStatus := SHL(BOOL_TO_DWORD(StrPh.error), PhaseNumber);
  StrPh.topStatus := SHL(BOOL_TO_DWORD(StrPh.top), PhaseNumber);
END_FUNCTION_BLOCK

FUNCTION_BLOCK fb_ph_OilPump
  VAR_IN_OUT
    im : struct_OilPump;
  END_VAR
  VAR_INPUT
    act : TYPE_DualStateImAction;
    PhaseNumber : UINT;
  END_VAR
  VAR_IN_OUT
    StrPh : struct_PhaseAlgoritm;
  END_VAR
  VAR
    CommandFault_Trig : R_TRIG;
    reset_Trig : R_TRIG;
    _statusDualInput : TYPE_statusDualInput;
  END_VAR

  IF StrPh.run AND NOT StrPh.start THEN
  	StrPh.start := TRUE;
  	StrPh.top := FALSE;
  	StrPh.error := FALSE;

  	CASE act OF
  		(*DualStateImAction.on*)   _on :im.inOpcCommandsDisabled:=TRUE;
                                                      im.inCommand_Alg := 1; (*cmd_open*)
  		(*DualStateImAction.off*) _off :im.inOpcCommandsDisabled:=TRUE;
                                                      im.inCommand_Alg := 2; (*cmd_close*)
  	END_CASE;
  END_IF;

  IF StrPh.start OR StrPh.reset THEN
      StrPh.run:=FALSE;
  END_IF;

  IF StrPh.start AND NOT StrPh.top THEN
                      CommandFault_Trig(CLK := im.CommandFault);
                      IF CommandFault_Trig.Q THEN
  	          StrPh.error := TRUE;
                      END_IF;

  		CASE act OF
  		(*_DualStateImAction.on*)    _on: StrPh.top := im.onStatus = _statusDualInput.STATUS_ON;
  		(*_DualStateImAction.off*)  _off: StrPh.top := im.onStatus = _statusDualInput.STATUS_OFF;
  		END_CASE;

  END_IF;

  reset_Trig(CLK := StrPh.reset);
  IF reset_Trig.Q THEN
  	StrPh.start := FALSE;
  	StrPh.error := FALSE;
  	StrPh.top := FALSE;
            StrPh.reset:=FALSE;
  END_IF;

  StrPh.startStatus := SHL(BOOL_TO_DWORD(StrPh.start), PhaseNumber);
  StrPh.errorStatus := SHL(BOOL_TO_DWORD(StrPh.error), PhaseNumber);
  StrPh.topStatus := SHL(BOOL_TO_DWORD(StrPh.top), PhaseNumber);
END_FUNCTION_BLOCK

FUNCTION_BLOCK fb_sunpackerCommand
  VAR_INPUT
    command : WORD;
  END_VAR
  VAR_OUTPUT
    source : BYTE;
    parametr : BYTE;
    cmd : BYTE;
  END_VAR

  cmd := WORD_TO_BYTE(command and 16#7);
  parametr := WORD_TO_BYTE(SHR((command and 16#1FF8), 3));
  source := WORD_TO_BYTE(SHR(command, 13));
END_FUNCTION_BLOCK

FUNCTION resetIfRunningSO : BOOL
  VAR_IN_OUT
    so : struct_singleOutput;
  END_VAR
  VAR CONSTANT
    cmdReset : WORD          := 2;
  END_VAR

  IF so.Q THEN
                      so.inOpcCommandsDisabled:=TRUE;
  		so.inCommand_Alg:=cmdReset;
  END_IF;
END_FUNCTION

FUNCTION resetDiProtection : BOOL
  VAR_IN_OUT
    protection : struct_DiProtection;
  END_VAR
  VAR CONSTANT
    cmdReset : WORD          := 2;
  END_VAR

  IF protection.isRunning THEN
                      protection.inOpcCommandsDisabled:=TRUE;
  		protection.inCommand_Alg:=cmdReset;
  END_IF;
END_FUNCTION

FUNCTION resetAiProtection : BOOL
  VAR_IN_OUT
    protection : struct_AiProtection;
  END_VAR
  VAR CONSTANT
    cmdReset : WORD          := 2;
  END_VAR

  IF protection.isRunning THEN
                      protection.inOpcCommandsDisabled:=TRUE;
  		protection.inCommand_Alg:=cmdReset;
  END_IF;
END_FUNCTION

FUNCTION setValue : BOOL
  VAR_IN_OUT
    StrDP : struct_DiscretParametr;
  END_VAR
  VAR_INPUT
    newValue : UINT;
  END_VAR
  VAR
    cmd_ChangeValue : WORD          := 1;
  END_VAR

  StrDP.newValue:=newValue;
  StrDP.inOpcCommandsDisabled:=TRUE;
  StrDP.inCommand_Alg:=cmd_ChangeValue;
END_FUNCTION

FUNCTION runAiProtection : BOOL
  VAR_IN_OUT
    protection : struct_AiProtection;
  END_VAR
  VAR CONSTANT
    cmdRun : WORD          := 1;
  END_VAR

  IF NOT protection.isRunning THEN
                      protection.inOpcCommandsDisabled:=TRUE;
  		protection.inCommand_Alg:=cmdRun;
  END_IF;
END_FUNCTION

FUNCTION resetPhase : BOOL
  VAR_IN_OUT
    ph : struct_PhaseAlgoritm;
  END_VAR

  IF ph.start OR ph.top THEN
                      ph.reset:=TRUE;
  END_IF;
END_FUNCTION

FUNCTION impulseSO : BOOL
  VAR_IN_OUT
    so : struct_singleOutput;
  END_VAR
  VAR CONSTANT
    cmdImpulse : WORD          := 3;
  END_VAR

  IF NOT so.Q THEN
      so.inOpcCommandsDisabled:=TRUE;
      so.inCommand_Alg:=cmdImpulse;
  END_IF;
END_FUNCTION

FUNCTION runPhase : BOOL
  VAR_IN_OUT
    ph : struct_PhaseAlgoritm;
  END_VAR

  IF NOT ph.start THEN
                      ph.run:=TRUE;
  END_IF;
END_FUNCTION

FUNCTION runIfNotRunningSO : BOOL
  VAR_IN_OUT
    so : struct_singleOutput;
  END_VAR
  VAR CONSTANT
    cmdRun : WORD          := 1;
  END_VAR

  IF NOT so.Q THEN
                      so.inOpcCommandsDisabled:=TRUE;
  		so.inCommand_Alg:=cmdRun;
  END_IF;
END_FUNCTION

FUNCTION_BLOCK NOAlg
  VAR_IN_OUT
    StrAlg : struct_Alg;
  END_VAR
  VAR
    timer120 : struct_PhaseAlgoritm;
    kran6Open : struct_PhaseAlgoritm;
    pnsOn : struct_PhaseAlgoritm;
    kran4Close : struct_PhaseAlgoritm;
    kran3bOpen : struct_PhaseAlgoritm;
    mvOff : struct_PhaseAlgoritm;
    kran1Close : struct_PhaseAlgoritm;
    kran2Close : struct_PhaseAlgoritm;
    kran3Close : struct_PhaseAlgoritm;
    kran5Open : struct_PhaseAlgoritm;
    error_Krans : struct_PhaseAlgoritm;
    autoPnsOff : struct_PhaseAlgoritm;
    Pg_VhodLessThen300 : struct_PhaseAlgoritm;
    Pg_VyhodLessThen300 : struct_PhaseAlgoritm;
    nu1off : struct_PhaseAlgoritm;
    nu2off : struct_PhaseAlgoritm;
    AutoNU_Off : struct_PhaseAlgoritm;
    timer600 : struct_PhaseAlgoritm;
    pnsOff : struct_PhaseAlgoritm;
    Avom1Off : struct_PhaseAlgoritm;
    Avom2Off : struct_PhaseAlgoritm;
    Avom3Off : struct_PhaseAlgoritm;
    Avom4Off : struct_PhaseAlgoritm;
    autoAVOMOff : struct_PhaseAlgoritm;
    timer5 : struct_PhaseAlgoritm;
    klapan1 : struct_PhaseAlgoritm;
    klapan2 : struct_PhaseAlgoritm;
    nu_On : struct_PhaseAlgoritm;
    fb_timer120 : fb_ph_Timer;
    fb_kran6Open : fb_ph_Kran;
    fb_pnsOn : fb_ph_Switch;
    fb_kran4Close : fb_ph_Kran;
    fb_kran3bOpen : fb_ph_Kran;
    fb_mvOff : fb_ph_SectionSwitch;
    fb_kran1Close : fb_ph_Kran;
    fb_kran2Close : fb_ph_Kran;
    fb_kran3Close : fb_ph_Kran;
    fb_kran5Open : fb_ph_Kran;
    fb_error_Krans : fb_ph_CustomPhase;
    fb_autoPnsOff : fb_ph_algoritm;
    fb_Pg_VhodLessThen300 : fb_ph_CustomPhase;
    fb_Pg_VyhodLessThen300 : fb_ph_CustomPhase;
    fb_nu1Off : fb_ph_OilPump;
    fb_nu2Off : fb_ph_OilPump;
    fb_autoNuOff : fb_ph_algoritm;
    fb_timer600 : fb_ph_Timer;
    fb_pnsOff : fb_ph_Switch;
    fb_Avom1Off : fb_ph_Switch;
    fb_Avom2Off : fb_ph_Switch;
    fb_Avom3Off : fb_ph_Switch;
    fb_Avom4Off : fb_ph_Switch;
    fb_autoAVOMOff : fb_ph_algoritm;
    fb_timer5 : fb_ph_Timer;
    fb_klapan1 : fb_ph_CustomPhase;
    fb_klapan2 : fb_ph_CustomPhase;
    fb_nu_On : fb_ph_CustomPhase;
    _sunpackerCommand : fb_sunpackerCommand;
    _statusAi : TYPE_StatusAi;
    _Answers : TYPE_Answers;
    _statusDualInput : TYPE_statusDualInput;
    _commandDualInput : TYPE_commandDualInput;
    _DualStateImAction : TYPE_DualStateImAction;
    _PhaseAlgoritmAction : TYPE_PhaseAlgoritmAction;
    source : BYTE;
    cmd : BYTE;
    lastCmd : BYTE;
    source_for_Status : BYTE;
    cmd_for_Status : BYTE;
    command_error_for_Status : BYTE;
    resetCmdTimer : TON;
    resetCmdTimerPriznak : BOOL;
    onInit : BOOL;
    waitReset : TON;
  END_VAR
  VAR_EXTERNAL
    IM : ImConfig;
    algoritms : AlgoritmsConfig;
    ai : AiConfig;
    protections : ProtectionsConfig;
    ModeGpa : TYPE_ModeGpa;
    algManager : struct_AlgoritmsManager;
    AlgTimers : struct_AlgTimers;
  END_VAR
  VAR CONSTANT
    Ust_Pgaza : LREAL          := 0.3;
  END_VAR

  IF NOT onInit THEN
      fb_timer120(phaseNumber:=1, delay:=T#120S);
      fb_kran6Open(phaseNumber:=2, act:=_on);
      fb_kran4Close(phaseNumber:=3, act:=_off);
      fb_kran3bOpen(phaseNumber:=4, act:=_off);
      fb_mvOff(phaseNumber:=5, act:=_off);
      fb_kran1Close(phaseNumber:=6, act:=_off);
      fb_kran2Close(phaseNumber:=7, act:=_off);
      fb_kran3Close(phaseNumber:=8, act:=_off);
      fb_kran5Open(phaseNumber:=9, act:=_on);
      fb_error_Krans(phaseNumber:=10);
      fb_autoPnsOff(phaseNumber:=11, act:=_reset, waitCompletion:=FALSE);
      fb_pnsOn(phaseNumber:=12, act:=_on);
      fb_Pg_VhodLessThen300(phaseNumber:=13);
      fb_Pg_VyhodLessThen300(phaseNumber:=14);
      fb_nu1Off(phaseNumber:=15, act:=_off);
      fb_nu2Off(phaseNumber:=16, act:=_off);
      fb_autoNuOff(phaseNumber:=17, act:=_reset, waitCompletion:=FALSE);
      fb_timer600(phaseNumber:=18, delay:=T#600S);
      fb_pnsOff(phaseNumber:=19, act:=_off);
      fb_Avom1Off(phaseNumber:=20, act:=_off);
      fb_Avom2Off(phaseNumber:=21, act:=_off);
      fb_Avom3Off(phaseNumber:=22, act:=_off);
      fb_Avom4Off(phaseNumber:=23, act:=_off);
      fb_autoAVOMOff(phaseNumber:=24, act:=_reset, waitCompletion:=FALSE);
      fb_timer5(phaseNumber:=25, delay:=T#5S);
      fb_klapan1(phaseNumber:=26);
      fb_klapan2(phaseNumber:=27);
      fb_nu_On(phaseNumber:=28);

  onInit:=TRUE;
  END_IF;

  fb_timer120(StrPh:=timer120, timer:=AlgTimers.No_wait120);
  fb_kran6Open(StrPh:=kran6Open, Im:=Im.kran6);
  fb_pnsOn(StrPh:=pnsOn, Im:=Im.pns);
  fb_kran4Close(StrPh:=kran4Close, Im:=Im.kran4);
  fb_kran3bOpen(StrPh:=kran3bOpen, Im:=Im.kran3b);
  fb_mvOff(StrPh:=mvOff, Im:=Im.mv);
  fb_kran1Close(StrPh:=kran1Close, Im:=Im.kran1);
  fb_kran2Close(StrPh:=kran2Close, Im:=Im.Kran2);
  fb_kran3Close(StrPh:=kran3Close, Im:=Im.Kran3);
  fb_kran5Open(StrPh:=kran5Open, Im:=Im.Kran5);
  fb_error_Krans(StrPh:=error_Krans);
  fb_autoPnsOff(StrPh:=autoPnsOff, alg:=algoritms.autoPns);
  fb_Pg_VhodLessThen300(StrPh:=Pg_VhodLessThen300);
  fb_Pg_VyhodLessThen300(StrPh:=Pg_VyhodLessThen300);
  fb_nu1Off(StrPh:=nu1off, Im:=Im.nu1);
  fb_nu2Off(StrPh:=nu2off, Im:=Im.nu2);
  fb_autoNuOff(StrPh:=AutoNU_Off, alg:=algoritms.autoNu);
  fb_timer600(StrPh:=timer600, timer:=AlgTimers.No_wait600);
  fb_pnsOff(StrPh:=pnsOff, Im:=Im.pns);
  fb_Avom1Off(StrPh:=Avom1Off, Im:=Im.v1_Avom);
  fb_Avom2Off(StrPh:=Avom2Off, Im:=Im.v2_Avom);
  fb_Avom3Off(StrPh:=Avom3Off, Im:=Im.v3_Avom);
  fb_Avom4Off(StrPh:=Avom4Off, Im:=Im.v4_Avom);
  fb_autoAVOMOff(StrPh:=autoAVOMOff, alg:=algoritms.AutoAvom);
  fb_timer5(StrPh:=timer5, timer:=AlgTimers.No_wait5);
  fb_klapan1(StrPh:=klapan1);
  fb_klapan2(StrPh:=klapan2);
  fb_nu_On(StrPh:=nu_On);

  StrAlg.CanRun := StrAlg.inCanRun;
  StrAlg.OpcCommandsDisabled := StrAlg.inOpcCommandsDisabled;

  IF StrAlg.isRuning THEN
      (* кран 6 не открыт - запуск таймера *)
      IF NOT kran6Open.top AND NOT timer120.top  THEN
  	runPhase(timer120);
      ELSE
      (* счетчик отработал и кран 6 не открыт - ошибка *)
          IF timer120.top AND NOT kran6Open.top THEN
              error_Krans.error := TRUE;
          END_IF;
      END_IF;

      (* старт смазки кранов *)
      IF (*algoritms.F3.Smazka_1_2 OR *)IM.kran1.onStatus = _statusDualInput.STATUS_ON OR IM.kran1.onStatus = _statusDualInput.STATUS_TRANSITIONAL
  	OR IM.kran2.onStatus = _statusDualInput.STATUS_ON OR IM.kran2.onStatus = _statusDualInput.STATUS_TRANSITIONAL  THEN
          IF (*(algoritms.F3.Smazka_1_2 OR *)IM.kran1.onStatus = _statusDualInput.STATUS_ON OR IM.kran1.onStatus = _statusDualInput.STATUS_TRANSITIONAL AND NOT klapan1.start AND NOT kran1Close.top THEN
              runPhase(klapan1);
          END_IF;
          IF (*(algoritms.F3.Smazka_1_2 OR *)IM.kran2.onStatus = _statusDualInput.STATUS_ON OR IM.kran2.onStatus = _statusDualInput.STATUS_TRANSITIONAL AND NOT klapan2.start AND NOT kran2Close.top THEN
              runPhase(klapan2);
          END_IF;
      (*algoritms.F3.Smazka_1_2:=FALSE;*)
      END_IF;

      (* открыть кран 6 кран 4 *)
      runPhase(kran6Open);
      runPhase(kran4Close);

      (*не понимаю
      IF kran4Close.top THEN
          ystavki.Block_kr4_alg.setValue (0);
      END_IF;*)

      (* кран 6 открыт *)
      IF kran6Open.top THEN
  	runPhase(kran3bOpen);
  	resetPhase(timer120);
  	(*error_Krans.top := FALSE;
  	error_Krans.error := FALSE;*)
  	(*algoritms.S_Vibr.CanRun:=FALSE;
  	algoritms.S_Vibr.reset (); net takogo alg*)
      END_IF;
      IF kran3bOpen.top AND NOT mvoff.start THEN
  	resetDiProtection(protections.mvOff);
  	resetDiProtection(protections.Off_avar_vikluchatel);
  	resetDiProtection(protections.Reg_vozb_off);
  	runPhase(mvOff);
      END_IF;

      IF mvOff.top (*AND NOT flag1*) THEN
          algoritms.AutoPns.inCanRun :=FALSE;
          (*algoritms.AutoPNS_Start.reset (); nichego ne ponimau
          algoritms.AutoPns.inCanRun :=FALSE;*)
          runPhase(autoPnsOff);
          runPhase(pnsOn);
          resetDiProtection(protections.Kran1_sdvig);
          resetDiProtection(protections.Kran2_sdvig);
          runPhase(kran1Close);
          runPhase(kran2Close);
          runPhase(kran3Close);
          runPhase(nu_On);

          (*тут запустить насосы уплотнения *)

          (*algoritms.autoNu.inCanRun:=FALSE;
          algoritms.autoNu_2.reset ();
          algoritms.autoNu_1.inCanRun:=TRUE;
          algoritms.autoNu_1.run ();
          flag1:=TRUE; что тут происходит?*)
      END_IF;
      IF ((IM.nu1.onStatus =_statusDualInput.STATUS_ON) OR (IM.nu2.onStatus =_statusDualInput.STATUS_ON)) AND nu_On.start AND NOT nu_On.top THEN
          nu_On.top:=TRUE;
      END_IF;

      (* выдача смазки *)
      IF klapan1.start AND kran1Close.top THEN
          (*IM.Kr1_Smazka.impulse(); не понимаю((((((((*)
          klapan1.top:=TRUE;
      END_IF;

      IF klapan2.start AND kran2Close.top THEN
  	(*IM.Kr2_Smazka.impulse(); не понимаю *)
  	klapan2.top:=TRUE;
      END_IF;

      (* кран 1 кран 2 кран 3 кран 4 закрыты - открыть кран 5 *)
      IF kran1Close.top AND kran2Close.top AND kran3Close.top AND kran4Close.top THEN
          runPhase(kran5Open);
          resetAiProtection(protections.Pgaza_na_vyhode_nagnetatelia);
      END_IF;

      IF kran5Open.top THEN
          runPhase(Pg_VhodLessThen300);
          runPhase(Pg_VyhodLessThen300);
      END_IF;

      IF Pg_VhodLessThen300.start AND NOT Pg_VhodLessThen300.top THEN
          IF (ai.Pgaza_na_vhode_nagnetatelia.interval>= _statusAi.NORMAL) AND (ai.Pgaza_na_vhode_nagnetatelia.value < 0.3) THEN
              Pg_VhodLessThen300.top:=TRUE;
          END_IF;
      END_IF;

      IF Pg_VyhodLessThen300.start AND NOT Pg_VyhodLessThen300.top THEN
          IF (ai.Pgaza_na_vyhode_nagnetatelia.interval>=_statusAi.NORMAL) AND (ai.Pgaza_na_vyhode_nagnetatelia.value < 0.3) THEN
              Pg_VyhodLessThen300.top:=TRUE;
          END_IF;
      END_IF;

      IF Pg_VhodLessThen300.top AND Pg_VyhodLessThen300.top AND pnsOn.top AND nu_On.top AND mvOff.top  THEN
          runphase(nu1Off);
          runphase(nu2Off);

          resetAiProtection(protections.dPmaslo_gaz);
          resetDiProtection(protections.dPmaslo_gaz_less100);

          runAiProtection(protections.Pgaza_na_vyhode_nagnetatelia_GPA_STOP);
          runAiProtection(protections.Pgaza_na_vhode_nagnetatelia_GPA_STOP);
          algoritms.autoNu.CanRun:=FALSE;
          AutoNU_Off.top:=TRUE;
          (*algoritms.autoNu_1.reset(); кого, чего куда*)
      END_IF;

      IF nu1Off.top THEN
          IF (*NOT algManager.reg_V AND кто чего*) NOT pnsoff.start THEN
              runPhase(timer600);
          END_IF;
          (*IF NOT pnsoff.start THEN
              sbrosVibeg.ask();
          END_IF; kto chego?*)
      END_IF;

      IF timer600.top (*OR sbrosVibeg.answer=Answers.ANS_YES kto chto *)THEN
  	runPhase(pnsOff);
  	resetAiProtection(protections.Pmaslo_sm_nizkoe);
  	resetAiProtection(protections.Pmaslo_sm_vysokoe);
  	(*sbrosVibeg.reset (); pomogite *)
  	resetPhase(timer600);
  	(*algoritms.F2_Ch.autoAVOM_canrun_flag:=FALSE;
  	algoritms.F2_R.autoAVOM_canrun_flag:=FALSE;*)
      END_IF;
      IF (*(NOT algoritms.F2_Ch.autoAVOM_canrun_flag) AND (NOT algoritms.F2_R.autoAVOM_canrun_flag) AND*)pnsoff.start THEN
  	runPhase(Avom1Off);
  	runPhase(Avom2Off);
  	runPhase(Avom3Off);
  	runPhase(Avom4Off);

  	(*algoritms.R_AutoAVOM.CanRun:=FALSE;
  	algoritms.R_AutoAVOM.reset();
  	algoritms.S_AutoAVOM.CanRun:=FALSE;
  	algoritms.S_AutoAVOM.reset();
  	algoritms.Auto_Avom_.CanRun:=FALSE;*)
  	runPhase(autoAVOMOff);
      END_IF;

      IF pnsOff.top AND Avom1Off.top AND Avom2Off.top AND Avom3Off.top AND Avom4Off.top AND autoAVOMOff.top  THEN
          runPhase(timer5);
      END_IF;

      IF timer5.top THEN
  	resetPhase(timer5);
      END_IF;
  END_IF;

  _sunpackerCommand(command := StrAlg.inCommand);
  	source := _sunpackerCommand.source;
  	cmd := _sunpackerCommand.cmd;

  IF cmd <> 0 AND lastCmd <> cmd AND (((NOT StrAlg.opcCommandsDisabled) AND source > 0) OR source = 0) then
  	CASE BYTE_TO_INT(cmd) OF
  		(*cmdRun*) 1: 	IF (StrAlg.CanRun) THEN
  					StrAlg.isRuning := TRUE;
  					StrAlg.isEnded := FALSE;
  					StrAlg.hasError := FALSE;
  					(*****************       OnRun       *****************)

                                                    algManager.nMode:=ModeGpa.MODE_NO;
                                                    (*runIfNotRunningSO(IM.SingleOutputs.Lampa_NO);*)

                                                    runPhase(kran4Close);
                                                    runPhase(timer120);
                                                    runPhase(nu1Off);
                                                    runPhase(timer600);

                                                   (* resetAiProtection(protections.Pgaza_na_vyhode_nagnetatelia);
                                                    resetAiProtection(protections.dPmaslo_gaz);
                                                    resetAiProtection(protections.Pmaslo_sm_nizkoe);
                                                    resetAiProtection(protections.Pmaslo_sm_vysokoe);
                                                    resetAiProtection(protections.Pgaza_na_vhode_nagnetatelia);
                                                    resetAiProtection(protections.Pgaza_na_vyhode_nagnetatelia);
                                                    resetDiProtection(protections.Reg_vozb_off);
                                                    resetDiProtection(protections.Fail_chastotnii_pusk);*)

  					cmd_for_Status := cmd;
  					source_for_Status := source;
  					command_error_for_Status := 0;
  				ELSE
  					StrAlg.isRuning := FALSE;
  					StrAlg.isEnded := FALSE;
  					StrAlg.hasError 	:= FALSE;

  					cmd_for_Status := 0;
  					source_for_Status := source;
  					command_error_for_Status := cmd;
  				END_IF;
  		(*cmdReset*) 2: 	StrAlg.isRuning := FALSE;
  				StrAlg.isEnded := FALSE;
  				StrAlg.hasError 	:= FALSE;

                                           (*****************       OnReset       *****************)
                                          waitReset(IN:=FALSE);
                                          (*resetIfRunningSO(IM.SingleOutputs.Lampa_NO);*)
                                          resetIfRunning(algoritms.vibegPNS);
                                          (*impulseSO(Im.SingleOutputs.SbrosBREO);*)

                                          resetPhase(timer120);
                                          resetPhase(kran6Open);
                                          resetPhase(pnsOn);
                                          resetPhase(kran4Close);
                                          resetPhase(kran3bOpen);
                                          resetPhase(mvOff);
                                          resetPhase(kran1Close);
                                          resetPhase(kran2Close);
                                          resetPhase(kran3Close);
                                          resetPhase(kran5Open);
  	                              resetPhase(error_Krans);
                                          resetPhase(autoPnsOff);
                                          resetPhase(pnsOn);
                                          resetPhase(Pg_VhodLessThen300);
                                          resetPhase(Pg_VyhodLessThen300);
                                          resetPhase(nu2Off);
                                          resetPhase(nu1Off);
                                          resetPhase(AutoNU_Off);
                                          resetPhase(timer600);

  				cmd_for_Status := cmd;
  				source_for_Status := source;
  				command_error_for_Status := 0;
  	END_CASE;
  	resetCmdTimer(IN := false);
  	resetCmdTimerPriznak := TRUE;
  END_IF;
  lastCmd := cmd;

  resetCmdTimer(IN := resetCmdTimerPriznak, PT := T#5S);
  IF resetCmdTimer.Q THEN
  	resetCmdTimerPriznak := FALSE;
  	source_for_Status := 0;
  	cmd_for_Status := 0;
  	command_error_for_Status := 0;
  END_IF;

  StrAlg.Start:= timer120.startStatus
              OR kran6Open.startStatus
              OR pnsOn.startStatus
              OR kran4Close.startStatus
              OR kran3bOpen.startStatus
              OR mvOff.startStatus
              OR kran1Close.startStatus
              OR kran2Close.startStatus
              OR kran3Close.startStatus
              OR kran5Open.startStatus
              OR error_Krans.startStatus
              OR autoPnsOff.startStatus
              OR pnsOn.startStatus
              OR Pg_VhodLessThen300.startStatus
              OR Pg_VyhodLessThen300.startStatus
              OR nu2Off.startStatus
              OR nu1Off.startStatus
              OR AutoNU_Off.startStatus
              OR timer600.startStatus;

  StrAlg.Error:= timer120.errorStatus
              OR kran6Open.errorStatus
              OR pnsOn.errorStatus
              OR kran4Close.errorStatus
              OR kran3bOpen.errorStatus
              OR mvOff.errorStatus
              OR kran1Close.errorStatus
              OR kran2Close.errorStatus
              OR kran3Close.errorStatus
              OR kran5Open.errorStatus
              OR error_Krans.errorStatus
              OR autoPnsOff.errorStatus
              OR pnsOn.errorStatus
              OR Pg_VhodLessThen300.errorStatus
              OR Pg_VyhodLessThen300.errorStatus
              OR nu2Off.errorStatus
              OR nu1Off.errorStatus
              OR AutoNU_Off.errorStatus
              OR timer600.errorStatus;

  StrAlg.Top:=   timer120.topStatus
              OR kran6Open.topStatus
              OR pnsOn.topStatus
              OR kran4Close.topStatus
              OR kran3bOpen.topStatus
              OR mvOff.topStatus
              OR kran1Close.topStatus
              OR kran2Close.topStatus
              OR kran3Close.topStatus
              OR kran5Open.topStatus
              OR error_Krans.topStatus
              OR autoPnsOff.topStatus
              OR pnsOn.topStatus
              OR Pg_VhodLessThen300.topStatus
              OR Pg_VyhodLessThen300.topStatus
              OR nu2Off.topStatus
              OR nu1Off.topStatus
              OR AutoNU_Off.topStatus
              OR timer600.topStatus;

  (*TODO: TYPE PROGRAM CODE HERE*)
  StrAlg.status :=  SHL(BYTE_TO_DWORD(source_for_Status), 29)
  			OR SHL(BYTE_TO_DWORD(cmd_for_Status), 26)
  			OR SHL(BYTE_TO_DWORD(command_error_for_Status), 23)
  			OR SHL(BOOL_TO_DWORD(StrAlg.OpcCommandsDisabled ), 21)
  			OR SHL(BOOL_TO_DWORD(StrAlg.hasError),4)
  			OR SHL(BOOL_TO_DWORD(StrAlg.CanRun),2)
  			OR SHL(BOOL_TO_DWORD(StrAlg.isEnded),1)
  			OR BOOL_TO_DWORD(StrAlg.isRuning);
END_FUNCTION_BLOCK

FUNCTION runDiProtection : BOOL
  VAR_IN_OUT
    protection : struct_DiProtection;
  END_VAR
  VAR CONSTANT
    cmdRun : WORD          := 1;
  END_VAR

  IF NOT protection.isRunning THEN
                      protection.inOpcCommandsDisabled:=TRUE;
  		protection.inCommand_Alg:=cmdRun;
  END_IF;
END_FUNCTION

FUNCTION_BLOCK fb_ph_DIprotection
  VAR_IN_OUT
    StrDiP : struct_DiProtection;
  END_VAR
  VAR_INPUT
    act : TYPE_PhaseAlgoritmAction;
    PhaseNumber : UINT;
  END_VAR
  VAR_IN_OUT
    StrPh : struct_PhaseAlgoritm;
  END_VAR
  VAR
    CommandFault_Trig : R_TRIG;
    reset_Trig : R_TRIG;
    _statusDualInput : TYPE_statusDualInput;
  END_VAR

  IF StrPh.run AND NOT StrPh.start THEN
  	StrPh.start := TRUE;
  	StrPh.top := FALSE;
  	StrPh.error := FALSE;
            StrPh.run:=FALSE;

  	CASE act OF
  		(*PhaseAlgoritmAction.run*)    _run : runDiProtection(StrDiP); (*cmd_run*)
  		(*PhaseAlgoritmAction.reset*)_reset : resetDiProtection(StrDiP); (*cmd_reset*)
  	END_CASE;
  END_IF;

  IF StrPh.start AND NOT StrPh.top THEN
                      CommandFault_Trig(CLK := StrDiP.hasError);
                      IF CommandFault_Trig.Q THEN
  	          StrPh.error := TRUE;
                      END_IF;

  		CASE act OF
  		(*PhaseAlgoritmAction.run*)    _run:    StrPh.top:=StrDiP.isRunning;

  		(*PhaseAlgoritmAction.reset*) _reset:   StrPh.top := NOT StrDiP.isRunning;
  		END_CASE;

  END_IF;

  IF StrPh.top THEN
  StrPh.error := FALSE;
  END_IF;

  reset_Trig(CLK := StrPh.reset);
  IF reset_Trig.Q THEN
            StrPh.start := FALSE;
  	StrPh.error := FALSE;
  	StrPh.top := FALSE;
            StrPh.run:=FALSE;
            StrPh.reset:=FALSE;
  END_IF;

  StrPh.startStatus := SHL(BOOL_TO_DWORD(StrPh.start), PhaseNumber);
  StrPh.errorStatus := SHL(BOOL_TO_DWORD(StrPh.error), PhaseNumber);
  StrPh.topStatus := SHL(BOOL_TO_DWORD(StrPh.top), PhaseNumber);
END_FUNCTION_BLOCK

FUNCTION_BLOCK fillingAlg
  VAR_IN_OUT
    StrAlg : struct_Alg;
  END_VAR
  VAR
    BreakPuskTimer : struct_PhaseAlgoritm;
    kran3bOpen : struct_PhaseAlgoritm;
    kran4Open : struct_PhaseAlgoritm;
    waitAfterKran4 : struct_PhaseAlgoritm;
    kran5Close : struct_PhaseAlgoritm;
    didPKran1 : struct_PhaseAlgoritm;
    kran1Open : struct_PhaseAlgoritm;
    kran2Open : struct_PhaseAlgoritm;
    kran3bClose : struct_PhaseAlgoritm;
    kran4Close : struct_PhaseAlgoritm;
    RunProtection_kr1 : struct_PhaseAlgoritm;
    RunProtection_kr2 : struct_PhaseAlgoritm;
    waitAfterKran5 : struct_PhaseAlgoritm;
    testUnsuccessfulFilling : struct_PhaseAlgoritm;
    fb_BreakPuskTimer : fb_ph_Timer;
    fb_kran3bOpen : fb_ph_Kran;
    fb_kran4Open : fb_ph_Kran;
    fb_waitAfterKran4 : fb_ph_Timer;
    fb_kran5Close : fb_ph_Kran;
    fb_didPKran1 : fb_ph_CustomPhase;
    fb_kran1Open : fb_ph_Kran;
    fb_kran2Open : fb_ph_Kran;
    fb_kran3bClose : fb_ph_Kran;
    fb_kran4Close : fb_ph_Kran;
    fb_RunProtection_kr1 : fb_ph_DIprotection;
    fb_RunProtection_kr2 : fb_ph_DIprotection;
    fb_waitAfterKran5 : fb_ph_Timer;
    fb_testUnsuccessfulFilling : fb_ph_CustomPhase;
    _sunpackerCommand : fb_sunpackerCommand;
    _DualStateImAction : TYPE_DualStateImAction;
    _PhaseAlgoritmAction : TYPE_PhaseAlgoritmAction;
    source : BYTE;
    cmd : BYTE;
    lastCmd : BYTE;
    source_for_Status : BYTE;
    cmd_for_Status : BYTE;
    command_error_for_Status : BYTE;
    resetCmdTimer : TON;
    resetCmdTimerPriznak : BOOL;
    onInit : BOOL;
    waitReset : TON;
  END_VAR
  VAR_EXTERNAL
    IM : ImConfig;
    ai : AiConfig;
    protections : ProtectionsConfig;
    AlgTimers : struct_AlgTimers;
    algoritms : AlgoritmsConfig;
  END_VAR

  IF NOT onInit THEN

           fb_BreakPuskTimer(phaseNumber:=0, delay:=T#240S);
               fb_kran3bOpen(phaseNumber:=1, act:=_on);
                fb_kran4Open(phaseNumber:=2, act:=_on);
           fb_waitAfterKran4(phaseNumber:=3, delay:=T#10S);
               fb_kran5Close(phaseNumber:=4, act:=_off);
                fb_didPKran1(phaseNumber:=5);
                fb_kran1Open(phaseNumber:=7, act:=_on);
                fb_kran2Open(phaseNumber:=8, act:=_on);
              fb_kran3bClose(phaseNumber:=9, act:=_off);
               fb_kran4Close(phaseNumber:=10, act:=_off);
        fb_RunProtection_kr1(phaseNumber:=11, act:=_run);
        fb_RunProtection_kr2(phaseNumber:=12, act:=_run);
           fb_waitAfterKran5(phaseNumber:=13, delay:=T#60S);
  fb_testUnsuccessfulFilling(phaseNumber:=17);

  onInit:=TRUE;
  END_IF;

           fb_BreakPuskTimer(StrPh:=BreakPuskTimer, timer:=AlgTimers.filling_BreakPuskTimer);
               fb_kran3bOpen(StrPh:=kran3bOpen, Im:=Im.kran3b);
                fb_kran4Open(StrPh:=kran4Open, Im:=Im.kran4);
           fb_waitAfterKran4(StrPh:=waitAfterKran4, timer:=AlgTimers.filling_waitAfterKran4);
               fb_kran5Close(StrPh:=kran5Close, Im:=Im.kran5);
                fb_didPKran1(StrPh:=didPKran1);
                fb_kran1Open(StrPh:=kran1Open, Im:=Im.kran1);
                fb_kran2Open(StrPh:=kran2Open, Im:=Im.kran2);
              fb_kran3bClose(StrPh:=kran3bClose, Im:=Im.kran3b);
               fb_kran4Close(StrPh:=kran4Close, Im:=Im.kran4);
        fb_RunProtection_kr1(StrPh:=RunProtection_kr1 , StrDiP:=protections.Reg_vozb_off);
        fb_RunProtection_kr2(StrPh:=RunProtection_kr2 , StrDiP:=protections.Fail_chastotnii_pusk);
           fb_waitAfterKran5(StrPh:=waitAfterKran5, timer:=AlgTimers.filling_waitAfterKran5);
  fb_testUnsuccessfulFilling(StrPh:=testUnsuccessfulFilling);

  StrAlg.CanRun := StrAlg.inCanRun;
  StrAlg.OpcCommandsDisabled := StrAlg.inOpcCommandsDisabled;

  IF StrAlg.isRuning THEN

      StrAlg.hasError := kran3bOpen.error OR kran4Open.error OR kran5Close.error OR kran5Close.error
      OR kran1Open.error OR kran2Open.error OR kran3bClose.error OR kran4Close.error OR testUnsuccessfulFilling.error;

      IF kran4Open.top THEN
          runPhase(waitAfterKran4);
      END_IF;

      IF waitAfterKran4.top THEN
          runPhase(kran5Close);
      END_IF;

      IF kran3bOpen.top AND kran5Close.top THEN
         runPhase(waitAfterKran5);
         runPhase(didPKran1);
      END_IF;

      (*IF didPKran1.start AND NOT didPKran1.top THEN
      didPKran1.top:= im.singleSignals.dP_gazgaz_Kran1.Q;
      END_IF;*)

      IF waitAfterKran5.top AND didPKran1.top THEN
            runPhase(kran1Open);
  	runPhase(kran2Open);
      END_IF;

      IF kran1Open.top AND kran2Open.top THEN
            runPhase(kran4Close);
  	runPhase(kran3bClose);
      END_IF;

      IF kran4Close.top AND kran3bClose.top THEN

            runPhase(RunProtection_kr1);
            runPhase(RunProtection_kr2);

            (*runAiProtection(protections.Pgaza_na_vhode_nagnetatelia);
            runAiProtection(protections.Pgaza_na_vhode_nagnetatelia);
            runAiProtection(protections.Pgaza_na_vyhode_nagnetatelia);
            runAiProtection(protections.dPmaslo_gaz);
            runAiProtection(protections.Pmaslo_sm_nizkoe);
            runAiProtection(protections.Pmaslo_sm_vysokoe);*)

      END_IF;

      IF BreakPuskTimer.top AND NOT (RunProtection_kr1.top AND RunProtection_kr2.top ) THEN
  	testUnsuccessfulFilling.error:=TRUE;
      END_IF;

      IF RunProtection_kr1.top AND RunProtection_kr2.top THEN
            resetPhase(BreakPuskTimer);
  	waitReset(IN:=TRUE, PT:= T#2S);
      END_IF;

      IF waitReset.Q AND NOT (algoritms.Apusk.isRuning OR algoritms.SemiAutoPusk.isRuning) THEN
  	resetIfRunning(StrAlg);
      END_IF;

      StrAlg.isEnded:= RunProtection_kr1.top AND RunProtection_kr2.top;
  END_IF;

  StrAlg.CanRun := StrAlg.inCanRun;
  StrAlg.OpcCommandsDisabled := StrAlg.inOpcCommandsDisabled;

  (* ---- Если управление с ВУ заблокировано, то  передаем команду из алгоритма ---- *)
  IF StrAlg.inOpcCommandsDisabled THEN
  	StrAlg.inCommand := StrAlg.inCommand_Alg;
  ELSE (* иначе передаем команду с АРМа*)
  	StrAlg.inCommand := StrAlg.inCommand_ARM;
  END_IF;

  _sunpackerCommand(command := StrAlg.inCommand);
  	source := _sunpackerCommand.source;
  	cmd := _sunpackerCommand.cmd;

  IF cmd <> 0 AND lastCmd <> cmd AND (((NOT StrAlg.opcCommandsDisabled) AND source > 0) OR source = 0) then
  	CASE BYTE_TO_INT(cmd) OF
  		(*cmdRun*) 1: 	IF (StrAlg.CanRun) THEN
  					StrAlg.isRuning := TRUE;
  					StrAlg.isEnded := FALSE;
  					StrAlg.hasError := FALSE;
  					(*****************       OnRun       *****************)

                                                    runPhase(kran3bOpen);
                                                    runPhase(kran4Open);
                                                    runPhase(BreakPuskTimer);
                                                    runPhase(testUnsuccessfulFilling);

  					cmd_for_Status := cmd;
  					source_for_Status := source;
  					command_error_for_Status := 0;
  				ELSE
  					StrAlg.isRuning := FALSE;
  					StrAlg.isEnded := FALSE;
  					StrAlg.hasError 	:= FALSE;

  					cmd_for_Status := 0;
  					source_for_Status := source;
  					command_error_for_Status := cmd;
  				END_IF;
  		(*cmdReset*) 2: 	StrAlg.isRuning := FALSE;
  				StrAlg.isEnded := FALSE;
  				StrAlg.hasError 	:= FALSE;

                                           (*****************       OnReset       *****************)
                                          StrAlg.inCanRun:=FALSE;
                                          waitReset(IN:=FALSE);

                                          resetPhase(BreakPuskTimer);
                                          resetPhase(kran3bOpen);
                                          resetPhase(kran4Open);
                                          resetPhase(waitAfterKran4);
                                          resetPhase(kran5Close);
                                          resetPhase(didPKran1);
                                          resetPhase(kran1Open);
                                          resetPhase(kran2Open);
                                          resetPhase(kran3bClose);
                                          resetPhase(kran4Close);
  	                              resetPhase(RunProtection_kr1);
                                          resetPhase(RunProtection_kr2);
                                          resetPhase(waitAfterKran5);
                                          resetPhase(testUnsuccessfulFilling);

  				cmd_for_Status := cmd;
  				source_for_Status := source;
  				command_error_for_Status := 0;
  	END_CASE;
  	resetCmdTimer(IN := false);
  	resetCmdTimerPriznak := TRUE;
  END_IF;
  lastCmd := cmd;

  resetCmdTimer(IN := resetCmdTimerPriznak, PT := T#5S);
  IF resetCmdTimer.Q THEN
  	resetCmdTimerPriznak := FALSE;
  	source_for_Status := 0;
  	cmd_for_Status := 0;
  	command_error_for_Status := 0;
  END_IF;

  StrAlg.Start:= BreakPuskTimer.startStatus
              OR kran3bOpen.startStatus
              OR kran4Open.startStatus
              OR waitAfterKran4.startStatus
              OR kran5Close.startStatus
              OR didPKran1.startStatus
              OR kran1Open.startStatus
              OR kran2Open.startStatus
              OR kran3bClose.startStatus
              OR kran4Close.startStatus
              OR RunProtection_kr1.startStatus
              OR RunProtection_kr2.startStatus
              OR waitAfterKran5.startStatus
              OR testUnsuccessfulFilling.startStatus;

  StrAlg.Error:= BreakPuskTimer.errorStatus
              OR kran3bOpen.errorStatus
              OR kran4Open.errorStatus
              OR waitAfterKran4.errorStatus
              OR kran5Close.errorStatus
              OR didPKran1.errorStatus
              OR kran1Open.errorStatus
              OR kran2Open.errorStatus
              OR kran3bClose.errorStatus
              OR kran4Close.errorStatus
              OR RunProtection_kr1.errorStatus
              OR RunProtection_kr2.errorStatus
              OR waitAfterKran5.errorStatus
              OR testUnsuccessfulFilling.errorStatus;

  StrAlg.Top:=   BreakPuskTimer.topStatus
              OR kran3bOpen.topStatus
              OR kran4Open.topStatus
              OR waitAfterKran4.topStatus
              OR kran5Close.topStatus
              OR didPKran1.topStatus
              OR kran1Open.topStatus
              OR kran2Open.topStatus
              OR kran3bClose.topStatus
              OR kran4Close.topStatus
              OR RunProtection_kr1.topStatus
              OR RunProtection_kr2.topStatus
              OR waitAfterKran5.topStatus
              OR testUnsuccessfulFilling.topStatus;

  (*TODO: TYPE PROGRAM CODE HERE*)
  StrAlg.status :=  SHL(BYTE_TO_DWORD(source_for_Status), 29)
  			OR SHL(BYTE_TO_DWORD(cmd_for_Status), 26)
  			OR SHL(BYTE_TO_DWORD(command_error_for_Status), 23)
  			OR SHL(BOOL_TO_DWORD(StrAlg.OpcCommandsDisabled ), 21)
  			OR SHL(BOOL_TO_DWORD(StrAlg.hasError),4)
  			OR SHL(BOOL_TO_DWORD(StrAlg.CanRun),2)
  			OR SHL(BOOL_TO_DWORD(StrAlg.isEnded),1)
  			OR BOOL_TO_DWORD(StrAlg.isRuning);
END_FUNCTION_BLOCK

FUNCTION_BLOCK fb_singleSignal_Init
  VAR_INPUT
    data_Ini : BOOL;
    inverse : BOOL;
    DelayOn : TIME;
    DelayOff : TIME;
  END_VAR
  VAR_IN_OUT
    str_SS : struct_singleSignal;
  END_VAR
  VAR_OUTPUT
    Init : BOOL          := FALSE;
  END_VAR

  (*****            Функциональный блок переинициализации структуры  singleSignal          *****)
  Init := FALSE;

      IF data_Ini THEN                            (* Параметрам требуется переинициализация. *)
          str_SS.inverse                := inverse;
          str_SS.DelayOn                := DelayOn;
          str_SS.DelayOff               := DelayOff;

          data_Ini:=FALSE;
          Init := TRUE;
      END_IF;
   IF Init THEN
          inverse := FALSE;
          DelayOn := T#0S;
          DelayOff:= T#0S;
   END_IF;
END_FUNCTION_BLOCK

FUNCTION_BLOCK fb_singleSignal
  VAR_INPUT
    signal : TYPE_ReliableBit;
  END_VAR
  VAR_IN_OUT
    str_SS : struct_singleSignal;
  END_VAR
  VAR
    TimerOn : TON;
    TimerOff : TOF;
  END_VAR

  str_SS.reliability:=signal.reliability;

  IF NOT str_SS.inverse THEN
  TimerOn(IN:=(signal.value AND str_SS.reliability AND NOT str_SS.Disabled_Sig), PT:=str_SS.DelayOn);
  ELSE
  TimerOn(IN:=(signal._inversed AND str_SS.reliability AND NOT str_SS.Disabled_Sig), PT:=str_SS.DelayOn);
  END_IF;

  TimerOff(IN:=TimerOn.Q, PT:=str_SS.DelayOff);

  str_SS.Q:=TimerOff.Q;

  str_SS.status:= SHL(BOOL_TO_DWORD(NOT str_SS.reliability), 15)
  	OR BOOL_TO_DWORD(str_SS.Q);
END_FUNCTION_BLOCK

FUNCTION_BLOCK fb_MvProtection
  VAR_INPUT
    sw : struct_SectionSwitch;
  END_VAR
  VAR_IN_OUT
    StrDIp : struct_DiProtection;
  END_VAR
  VAR
    _sunpackerCommand : fb_sunpackerCommand;
    statusDualInput : TYPE_statusDualInput;
    _ProtectionTags : TYPE_ProtectionTags;
    _signalingTp : TOF;
    timer : TON;
    SignalingTrig : R_TRIG;
    SignalingFTrig : F_TRIG;
    SignalingDi : BOOL;
    source : BYTE;
    cmd : BYTE;
    lastCmd : BYTE;
    source_for_Status : BYTE;
    cmd_for_Status : BYTE;
    command_error_for_Status : BYTE;
    resetCmdTimer : TON;
    resetCmdTimerPriznak : BOOL;
    signalinTimer : TON;
    runOnStart_Trig : R_TRIG;
  END_VAR

  timer(IN := (sw.onStatus = statusDualInput.STATUS_OFF) AND StrDIp.isRunning  , PT := StrDIp.delay);
  SignalingTrig(CLK := timer.Q);
  IF SignalingTrig.Q THEN
  	SignalingDi := TRUE;
  END_IF;
  SignalingFTrig(CLK := timer.Q);
  IF SignalingFTrig.Q THEN
  	SignalingDi := FALSE;
  END_IF;

  StrDIp.Tag := StrDIp.inTag;
  StrDIp.RunOnStart := StrDIp.inRunOnStart;

  StrDIp.CanRun := StrDIp.inCanRun;

  StrDIp.OpcCommandsDisabled := StrDIp.inOpcCommandsDisabled;

  (* ---- Если управление с ВУ заблокировано, то передаем команду из алгоритма ---- *)
  IF StrDIp.inOpcCommandsDisabled THEN
  	StrDIp.inCommand := StrDIp.inCommand_Alg;
  ELSE (* иначе передаем команду с АРМа*)
  	StrDIp.inCommand := StrDIp.inCommand_ARM;
  END_IF;

  _sunpackerCommand(command := StrDIp.inCommand);
  	source := _sunpackerCommand.source;
  	cmd := _sunpackerCommand.cmd;

  IF cmd <> 0 AND lastCmd <> cmd AND (((NOT StrDIp.opcCommandsDisabled) AND source > 0) OR source = 0) then
  	CASE BYTE_TO_INT(cmd) OF
  	        (*cmdRun*) 1: 	IF        NOT StrDIp.Remont THEN
  					StrDIp.isEnded := FALSE;
  					StrDIp.hasError 	:= FALSE;
  					StrDIp.isRunning := TRUE;
  					cmd_for_Status := cmd;
  					source_for_Status := source;
  					command_error_for_Status := 0;
  				ELSE
  					StrDIp.isRunning := FALSE;
  					StrDIp.isEnded := FALSE;
  					StrDIp.hasError 	:= FALSE;

  					cmd_for_Status := 0;
  					source_for_Status := source;
  					command_error_for_Status := cmd;
  				END_IF;
                                          StrDIp.inOpcCommandsDisabled:=FALSE;

                  (*cmdReset*) 2: 	StrDIp.isRunning := FALSE;
  				StrDIp.isEnded := FALSE;
  				StrDIp.hasError 	:= FALSE;
  				SignalingDi:= FALSE;
  				StrDIp.Check := FALSE;
  				cmd_for_Status := cmd;
  				source_for_Status := source;
  				command_error_for_Status := 0;
                                          StrDIp.inOpcCommandsDisabled:=FALSE;

  	(*cmd_setRemont*) 4 :	StrDIp.Remont := TRUE;
  				(*StrDIp.isRunning := FALSE;*)

  				cmd_for_Status := cmd;
  				source_for_Status := source;
  				command_error_for_Status := 0;

          (*cmd_resetRemont*) 5 : 	(*IF (sw.onStatus = statusDualInput.STATUS_OFF) THEN
  					cmd_for_Status := 0;
  					source_for_Status := 0;
  					command_error_for_Status := cmd;
  				ELSE*)
  					StrDIp.Remont := FALSE;
  					(*StrDIp.isRunning := TRUE;*)

  					cmd_for_Status := cmd;
  					source_for_Status := source;
  					command_error_for_Status := 0;
  				(*END_IF;*)

  	(*cmd_setCheck*) 6 : 	StrDIp.Check := TRUE;

  				cmd_for_Status := cmd;
  				source_for_Status := source;
  				command_error_for_Status := 0;
  	END_CASE;
  	resetCmdTimer(IN := false);
  	resetCmdTimerPriznak := TRUE;
  END_IF;
  lastCmd := cmd;

  resetCmdTimer(IN := resetCmdTimerPriznak);
  IF resetCmdTimer.Q THEN
  	resetCmdTimerPriznak := FALSE;
  	source_for_Status := 0;
  	cmd_for_Status := 0;
  	command_error_for_Status := 0;
  END_IF;

  IF StrDIp.isRunning AND  NOT StrDIp.Remont AND NOT StrDIp.Check THEN
  	StrDIp.Signaling := SignalingDi;
  	StrDIp.SignalingTP := _signalingTp.Q;
  ELSE
  	StrDIp.Signaling := 0;
  	StrDIp.SignalingTP := 0;
  END_IF;

  _signalingTp(in := StrDIp.Signaling, PT := T#1s);

  StrDIp.status :=  SHL(BYTE_TO_DWORD(source_for_Status), 29)
  			OR SHL(BYTE_TO_DWORD(cmd_for_Status), 26)
  			OR SHL(BYTE_TO_DWORD(command_error_for_Status), 23)
  			OR SHL(BOOL_TO_DWORD(StrDIp.OpcCommandsDisabled ), 21)
  			OR SHL(BOOL_TO_DWORD(StrDIp.Signaling), 16)
  			OR SHL(BOOL_TO_DWORD(StrDIp.RunOnStart ), 15)
  			OR SHL(BOOL_TO_DWORD(StrDIp.remont), 6)
  			OR SHL(BOOL_TO_DWORD(StrDIp.Check), 5)
  			OR SHL(BOOL_TO_DWORD(StrDIp.hasError), 4)
  			OR SHL(BOOL_TO_DWORD(StrDIp.SignalingTP), 3)
  			OR SHL(BOOL_TO_DWORD(StrDIp.CanRun), 2)
  			OR SHL(BOOL_TO_DWORD(StrDIp.isEnded), 1)
  			OR BOOL_TO_DWORD(StrDIp.isRunning);
END_FUNCTION_BLOCK

FUNCTION_BLOCK fb_meandr
  VAR
    _output : BOOL;
  END_VAR
  VAR_INPUT
    period : TIME          := T#300MS;
  END_VAR
  VAR
    timer : TON;
    FALSE_val : BOOL          := FALSE;
    TRUE_val : BOOL          := TRUE;
  END_VAR
  VAR_IN_OUT
    output : BOOL;
  END_VAR

  timer(in:=NOT FALSE_val,PT:=period);

  IF timer.Q THEN
      _output:=_output XOR TRUE_val;
      timer(in:=FALSE);
  END_IF;

  output:=_output;
END_FUNCTION_BLOCK

FUNCTION_BLOCK fb_DI_Init
  VAR_INPUT
    data_Ini : BOOL;
    imit : BOOL          := FALSE;
  END_VAR
  VAR_IN_OUT
    strDI : struct_DI;
  END_VAR
  VAR_OUTPUT
    Init : BOOL          := FALSE;
  END_VAR

  (*****            Функциональный блок переинициализации структуры-дескриптора канала дискретного ввода        *****)

   Init := FALSE;

      IF data_Ini THEN                            (* Параметрам требуется переинициализация. *)
          strDI.imit       := imit;
          data_Ini:=FALSE;
          Init := TRUE;
      END_IF;
    IF Init THEN
  imit:=FALSE;
      END_IF;
END_FUNCTION_BLOCK

FUNCTION_BLOCK fb_DiSourceMlp
  VAR_INPUT
    arDIN : TItemDIN;
    err_mod : TItemDIN;
  END_VAR
  VAR_IN_OUT
    strDI : struct_DI;
  END_VAR
  VAR_OUTPUT
    Bounce : BOOL;
  END_VAR
  VAR
    _value : WORD;
    _reliability : BOOL;
    bitNumber : INT;
    bitNum : INT;
  END_VAR

  strDI.blConnect := (*((UINT_TO_WORD(arDIN.wFlags) = 1472) and*) (UINT_TO_WORD(err_mod.wValue) = 20) and (UINT_TO_WORD(err_mod.wFlags) = 192);
  Bounce := (UINT_TO_WORD(arDIN.wFlags) AND 16#0020) <> 0;

  If NOT strDI.imit THEN
  _value:=UINT_TO_WORD(arDIN.wValue);

      IF strDI.blConnect THEN
            strDI.reliability:=0;
            strDI.value:=0;
  	FOR bitNumber:=0 TO 7 BY 1 DO

  		_reliability:=WORD_TO_BOOL(SHR(_value, bitNumber*2) AND 16#2);
  		strDI.reliability:=strDI.reliability OR SHL(BOOL_TO_WORD(_reliability),bitNumber);
  		IF _reliability THEN
  			strDI.value:=strDI.value OR SHL((SHR(_value, bitNumber*2) AND 16#1),bitNumber);
  		END_IF;
  	END_FOR;
      ELSE
  	strDI.reliability := 0;
      END_IF;

      FOR bitNum:=0 TO 15 BY 1 DO
  	          strDI.bits[bitNum].reliability :=WORD_TO_BOOL(SHR(strDI.reliability, bitNum) AND 16#1);
  	IF strDI.bits[bitNum].reliability THEN
  		strDI.bits[bitNum].value :=WORD_TO_BOOL(SHR(strDI.value, bitNum) AND 16#1);
                      strDI.bits[bitNum]._inversed :=NOT strDI.bits[bitNum].value;
  	END_IF;
      END_FOR;

  END_IF;
END_FUNCTION_BLOCK

FUNCTION_BLOCK ExtNarabotka
  VAR
    saveInterval : TIME          := T#30S;
    narabotka : UDINT;
    timer : RTC;
    saveTimer : TON;
  END_VAR
  VAR_IN_OUT
    retain_narabotka : UDINT;
  END_VAR
  VAR
    initialized : BOOL;
  END_VAR
  VAR_INPUT
    started : BOOL;
    reset : BOOL;
  END_VAR

  IF NOT initialized THEN
  	narabotka:=retain_narabotka;
  	initialized:=TRUE;
  END_IF;

  timer();

  IF timer.Q THEN
  	narabotka:=DT_TO_UDINT( timer.CDT);

  END_IF;
  saveTimer(IN:=TRUE, PT:=saveInterval);
  IF saveTimer.Q THEN
  	retain_narabotka:=narabotka;
  	saveTimer(IN:=FALSE);
  END_IF;

  IF started THEN
  	IF NOT timer.Q THEN
  		timer.PDT:=UDINT_TO_DT(narabotka);
                      timer.IN:=TRUE;
  	END_IF;
  ELSE
  	IF timer.Q THEN
  		timer.IN:=FALSE;
                      saveTimer.IN:=FALSE;
  	END_IF;
  END_IF;

  IF reset THEN
  timer.PDT:=UINT_TO_DT(0);
  IF timer.IN THEN
  	timer(IN:=FALSE);
  	timer(IN:=TRUE);
  END_IF;
  narabotka:=0;
  reset:=FALSE;
  END_IF;
END_FUNCTION_BLOCK

FUNCTION_BLOCK ph_SingleOutput
  VAR_IN_OUT
    im : struct_singleOutput;
  END_VAR
  VAR_INPUT
    WhatCanIdo : BOOL;
    PhaseNumber : UINT;
  END_VAR
  VAR_IN_OUT
    StrPh : struct_PhaseAlgoritm;
  END_VAR
  VAR
    reset_Trig : R_TRIG;
  END_VAR

  IF StrPh.run AND NOT StrPh.start THEN
  	StrPh.start := TRUE;
  	StrPh.top := FALSE;
  	StrPh.error := FALSE;
            StrPh.run:=FALSE;

  	IF (WhatCanIdo) THEN
  	runIfNotRunningSO(im);
            ELSE
  	resetIfRunningSO(im);
            END_IF;
  END_IF;

  IF StrPh.start AND NOT StrPh.top THEN
  StrPh.top := (im.Q = WhatCanIdo);
  END_IF;

  reset_Trig(CLK := StrPh.reset);
  IF reset_Trig.Q THEN
  	StrPh.start := FALSE;
  	StrPh.error := FALSE;
  	StrPh.top := FALSE;
            StrPh.run:=FALSE;
            StrPh.reset:=FALSE;
  END_IF;

  StrPh.startStatus := SHL(BOOL_TO_DWORD(StrPh.start), PhaseNumber);
  StrPh.errorStatus := SHL(BOOL_TO_DWORD(StrPh.error), PhaseNumber);
  StrPh.topStatus := SHL(BOOL_TO_DWORD(StrPh.top), PhaseNumber);
END_FUNCTION_BLOCK

FUNCTION_BLOCK OPC_PROTECTIONS_SET
  VAR_EXTERNAL
    protections : ProtectionsConfig;
    protections_Topornogo_podshipnika_EDT_1_inCommand_ARM : UINT;
    protections_Topornogo_podshipnika_EDT_1_status : UDINT;
    protections_Toy_podshipnika_EDT_2_inCommand_ARM : UINT;
    protections_Toy_podshipnika_EDT_2_status : UDINT;
    protections_Toy_podshipnika_kol_EDT_3_inCommand_ARM : UINT;
    protections_Toy_podshipnika_kol_EDT_3_status : UDINT;
    protections_Toy_podshipnika_kol_EDT_4_inCommand_ARM : UINT;
    protections_Toy_podshipnika_kol_EDT_4_status : UDINT;
    protections_To_podshipnika_shest_red_EDT_5_inCommand_ARM : UINT;
    protections_To_podshipnika_shest_red_EDT_5_status : UDINT;
    protections_To_podshipnika_shest_red_EDT_6_inCommand_ARM : UINT;
    protections_To_podshipnika_shest_red_EDT_6_status : UDINT;
    protections_To_podshipnika_N_EDT_7_inCommand_ARM : UINT;
    protections_To_podshipnika_N_EDT_7_status : UDINT;
    protections_To_podshipnika_svob_konca_EDT_8_inCommand_ARM : UINT;
    protections_To_podshipnika_svob_konca_EDT_8_status : UDINT;
    protections_Ty_podshipnika_rab_kol_EDT_9_inCommand_ARM : UINT;
    protections_Ty_podshipnika_rab_kol_EDT_9_status : UDINT;
    protections_Typornogo_podshipnika_nerab_kolodok_HT_10_inCommand_ARM : UINT;
    protections_Typornogo_podshipnika_nerab_kolodok_HT_10_status : UDINT;
    protections_Tgaza_na_vyhode_H_inCommand_ARM : UINT;
    protections_Tgaza_na_vyhode_H_status : UDINT;
    protections_Os_sdvig_nagnetatelja_plus_inCommand_ARM : UINT;
    protections_Os_sdvig_nagnetatelja_plus_status : UDINT;
    protections_Os_sdvig_nagnetatelja_minus_inCommand_ARM : UINT;
    protections_Os_sdvig_nagnetatelja_minus_status : UDINT;
    protections_Pgaza_na_vyhode_nagnetatelia_GPA_STOP_inCommand_ARM : UINT;
    protections_Pgaza_na_vyhode_nagnetatelia_GPA_STOP_status : UDINT;
    protections_Pgaza_na_vhode_nagnetatelia_GPA_STOP_inCommand_ARM : UINT;
    protections_Pgaza_na_vhode_nagnetatelia_GPA_STOP_status : UDINT;
    protections_Pgaza_na_vyhode_nagnetatelia_inCommand_ARM : UINT;
    protections_Pgaza_na_vyhode_nagnetatelia_status : UDINT;
    protections_dPmaslo_gaz_inCommand_ARM : UINT;
    protections_dPmaslo_gaz_status : UDINT;
    protections_Pmaslo_sm_nizkoe_inCommand_ARM : UINT;
    protections_Pmaslo_sm_nizkoe_status : UDINT;
    protections_Pmaslo_sm_vysokoe_inCommand_ARM : UINT;
    protections_Pmaslo_sm_vysokoe_status : UDINT;
    protections_Vibro_skorost_OPED_T1_inCommand_ARM : UINT;
    protections_Vibro_skorost_OPED_T1_status : UDINT;
    protections_Vibro_skorost_OPED_T2_inCommand_ARM : UINT;
    protections_Vibro_skorost_OPED_T2_status : UDINT;
    protections_Vibro_skorost_OYP_kolesa_ED_T3_inCommand_ARM : UINT;
    protections_Vibro_skorost_OYP_kolesa_ED_T3_status : UDINT;
    protections_Vibro_skorost_OP_kolesa_RH_T4_inCommand_ARM : UINT;
    protections_Vibro_skorost_OP_kolesa_RH_T4_status : UDINT;
    protections_Vibro_skorost_OP_shesterni_RED_T5_inCommand_ARM : UINT;
    protections_Vibro_skorost_OP_shesterni_RED_T5_status : UDINT;
    protections_Vibro_skorost_OP_shesterni_RED_T6_inCommand_ARM : UINT;
    protections_Vibro_skorost_OP_shesterni_RED_T6_status : UDINT;
    protections_dPmaslo_gaz_less100_inCommand_ARM : UINT;
    protections_dPmaslo_gaz_less100_status : UDINT;
    protections_Reg_vozb_off_inCommand_ARM : UINT;
    protections_Reg_vozb_off_status : UDINT;
    protections_Fail_chastotnii_pusk_inCommand_ARM : UINT;
    protections_Fail_chastotnii_pusk_status : UDINT;
    protections_Off_avar_vikluchatel_inCommand_ARM : UINT;
    protections_Off_avar_vikluchatel_status : UDINT;
    protections_AOKC_SHKC_inCommand_ARM : UINT;
    protections_AOKC_SHKC_status : UDINT;
    protections_AO_PRU_inCommand_ARM : UINT;
    protections_AO_PRU_status : UDINT;
    protections_AO_ot_SHU_inCommand_ARM : UINT;
    protections_AO_ot_SHU_status : UDINT;
    protections_mvOff_inCommand_ARM : UINT;
    protections_mvOff_status : UDINT;
    protections_Kran1_sdvig_inCommand_ARM : UINT;
    protections_Kran1_sdvig_status : UDINT;
    protections_Kran2_sdvig_inCommand_ARM : UINT;
    protections_Kran2_sdvig_status : UDINT;
  END_VAR

  protections_Topornogo_podshipnika_EDT_1_status := DWORD_TO_UDINT(protections.Topornogo_podshipnika_EDT_1.status);

      protections_Toy_podshipnika_EDT_2_status := DWORD_TO_UDINT(protections.Toy_podshipnika_EDT_2.status);

      protections_Toy_podshipnika_kol_EDT_3_status := DWORD_TO_UDINT(protections.Toy_podshipnika_kol_EDT_3.status);

      protections_Toy_podshipnika_kol_EDT_4_status := DWORD_TO_UDINT(protections.Toy_podshipnika_kol_EDT_4.status);

      protections_To_podshipnika_shest_red_EDT_5_status := DWORD_TO_UDINT(protections.To_podshipnika_shest_red_EDT_5.status);

      protections_To_podshipnika_shest_red_EDT_6_status := DWORD_TO_UDINT(protections.To_podshipnika_shest_red_EDT_6.status);

      protections_To_podshipnika_N_EDT_7_status := DWORD_TO_UDINT(protections.To_podshipnika_N_EDT_7.status);

      protections_To_podshipnika_svob_konca_EDT_8_status := DWORD_TO_UDINT(protections.To_podshipnika_svob_konca_EDT_8.status);

      protections_Ty_podshipnika_rab_kol_EDT_9_status := DWORD_TO_UDINT(protections.Ty_podshipnika_rab_kol_EDT_9.status);

      protections_Typornogo_podshipnika_nerab_kolodok_HT_10_status := DWORD_TO_UDINT(protections.Typornogo_podshipnika_nerab_kolodok_HT_10.status);

      protections_Tgaza_na_vyhode_H_status := DWORD_TO_UDINT(protections.Tgaza_na_vyhode_H.status);

      protections_Os_sdvig_nagnetatelja_plus_status := DWORD_TO_UDINT(protections.Os_sdvig_nagnetatelja_plus.status);

      protections_Os_sdvig_nagnetatelja_minus_status := DWORD_TO_UDINT(protections.Os_sdvig_nagnetatelja_minus.status);

      protections_Pgaza_na_vyhode_nagnetatelia_GPA_STOP_status := DWORD_TO_UDINT(protections.Pgaza_na_vyhode_nagnetatelia_GPA_STOP.status);

      protections_Pgaza_na_vhode_nagnetatelia_GPA_STOP_status := DWORD_TO_UDINT(protections.Pgaza_na_vhode_nagnetatelia_GPA_STOP.status);

      protections_Pgaza_na_vyhode_nagnetatelia_status := DWORD_TO_UDINT(protections.Pgaza_na_vyhode_nagnetatelia.status);

      protections_dPmaslo_gaz_status := DWORD_TO_UDINT(protections.dPmaslo_gaz.status);

      protections_Pmaslo_sm_nizkoe_status := DWORD_TO_UDINT(protections.Pmaslo_sm_nizkoe.status);

      protections_Pmaslo_sm_vysokoe_status := DWORD_TO_UDINT(protections.Pmaslo_sm_vysokoe.status);

      protections_Vibro_skorost_OPED_T1_status := DWORD_TO_UDINT(protections.Vibro_skorost_OPED_T1.status);

      protections_Vibro_skorost_OPED_T2_status := DWORD_TO_UDINT(protections.Vibro_skorost_OPED_T2.status);

      protections_Vibro_skorost_OYP_kolesa_ED_T3_status := DWORD_TO_UDINT(protections.Vibro_skorost_OYP_kolesa_ED_T3.status);

      protections_Vibro_skorost_OP_kolesa_RH_T4_status := DWORD_TO_UDINT(protections.Vibro_skorost_OP_kolesa_RH_T4.status);

      protections_Vibro_skorost_OP_shesterni_RED_T5_status := DWORD_TO_UDINT(protections.Vibro_skorost_OP_shesterni_RED_T5.status);

      protections_Vibro_skorost_OP_shesterni_RED_T6_status := DWORD_TO_UDINT(protections.Vibro_skorost_OP_shesterni_RED_T6.status);

      protections_dPmaslo_gaz_less100_status := DWORD_TO_UDINT(protections.dPmaslo_gaz_less100.status);

      protections_Reg_vozb_off_status := DWORD_TO_UDINT(protections.Reg_vozb_off.status);

      protections_Fail_chastotnii_pusk_status := DWORD_TO_UDINT(protections.Fail_chastotnii_pusk.status);

      protections_Off_avar_vikluchatel_status := DWORD_TO_UDINT(protections.Off_avar_vikluchatel.status);

      protections_AOKC_SHKC_status := DWORD_TO_UDINT(protections.AOKC_SHKC.status);

      protections_AO_PRU_status := DWORD_TO_UDINT(protections.AO_PRU.status);

      protections_AO_ot_SHU_status := DWORD_TO_UDINT(protections.AO_ot_SHU.status);

      protections_mvOff_status := DWORD_TO_UDINT(protections.mvOff.status);

      protections_Kran1_sdvig_status := DWORD_TO_UDINT(protections.Kran1_sdvig.status);

      protections_Kran2_sdvig_status := DWORD_TO_UDINT(protections.Kran2_sdvig.status);
END_FUNCTION_BLOCK

FUNCTION_BLOCK OPC_PROTECTIONS_GET
  VAR_EXTERNAL
    protections_Topornogo_podshipnika_EDT_1_inCommand_ARM : UINT;
    protections : ProtectionsConfig;
    protections_Topornogo_podshipnika_EDT_1_status : UDINT;
    protections_Toy_podshipnika_EDT_2_inCommand_ARM : UINT;
    protections_Toy_podshipnika_EDT_2_status : UDINT;
    protections_Toy_podshipnika_kol_EDT_3_inCommand_ARM : UINT;
    protections_Toy_podshipnika_kol_EDT_3_status : UDINT;
    protections_Toy_podshipnika_kol_EDT_4_inCommand_ARM : UINT;
    protections_Toy_podshipnika_kol_EDT_4_status : UDINT;
    protections_To_podshipnika_shest_red_EDT_5_inCommand_ARM : UINT;
    protections_To_podshipnika_shest_red_EDT_5_status : UDINT;
    protections_To_podshipnika_shest_red_EDT_6_inCommand_ARM : UINT;
    protections_To_podshipnika_shest_red_EDT_6_status : UDINT;
    protections_To_podshipnika_N_EDT_7_inCommand_ARM : UINT;
    protections_To_podshipnika_N_EDT_7_status : UDINT;
    protections_To_podshipnika_svob_konca_EDT_8_inCommand_ARM : UINT;
    protections_To_podshipnika_svob_konca_EDT_8_status : UDINT;
    protections_Ty_podshipnika_rab_kol_EDT_9_inCommand_ARM : UINT;
    protections_Ty_podshipnika_rab_kol_EDT_9_status : UDINT;
    protections_Typornogo_podshipnika_nerab_kolodok_HT_10_inCommand_ARM : UINT;
    protections_Typornogo_podshipnika_nerab_kolodok_HT_10_status : UDINT;
    protections_Tgaza_na_vyhode_H_inCommand_ARM : UINT;
    protections_Tgaza_na_vyhode_H_status : UDINT;
    protections_Os_sdvig_nagnetatelja_plus_inCommand_ARM : UINT;
    protections_Os_sdvig_nagnetatelja_plus_status : UDINT;
    protections_Os_sdvig_nagnetatelja_minus_inCommand_ARM : UINT;
    protections_Os_sdvig_nagnetatelja_minus_status : UDINT;
    protections_Pgaza_na_vyhode_nagnetatelia_GPA_STOP_inCommand_ARM : UINT;
    protections_Pgaza_na_vyhode_nagnetatelia_GPA_STOP_status : UDINT;
    protections_Pgaza_na_vhode_nagnetatelia_GPA_STOP_inCommand_ARM : UINT;
    protections_Pgaza_na_vhode_nagnetatelia_GPA_STOP_status : UDINT;
    protections_Pgaza_na_vyhode_nagnetatelia_inCommand_ARM : UINT;
    protections_Pgaza_na_vyhode_nagnetatelia_status : UDINT;
    protections_dPmaslo_gaz_inCommand_ARM : UINT;
    protections_dPmaslo_gaz_status : UDINT;
    protections_Pmaslo_sm_nizkoe_inCommand_ARM : UINT;
    protections_Pmaslo_sm_nizkoe_status : UDINT;
    protections_Pmaslo_sm_vysokoe_inCommand_ARM : UINT;
    protections_Pmaslo_sm_vysokoe_status : UDINT;
    protections_Vibro_skorost_OPED_T1_inCommand_ARM : UINT;
    protections_Vibro_skorost_OPED_T1_status : UDINT;
    protections_Vibro_skorost_OPED_T2_inCommand_ARM : UINT;
    protections_Vibro_skorost_OPED_T2_status : UDINT;
    protections_Vibro_skorost_OYP_kolesa_ED_T3_inCommand_ARM : UINT;
    protections_Vibro_skorost_OYP_kolesa_ED_T3_status : UDINT;
    protections_Vibro_skorost_OP_kolesa_RH_T4_inCommand_ARM : UINT;
    protections_Vibro_skorost_OP_kolesa_RH_T4_status : UDINT;
    protections_Vibro_skorost_OP_shesterni_RED_T5_inCommand_ARM : UINT;
    protections_Vibro_skorost_OP_shesterni_RED_T5_status : UDINT;
    protections_Vibro_skorost_OP_shesterni_RED_T6_inCommand_ARM : UINT;
    protections_Vibro_skorost_OP_shesterni_RED_T6_status : UDINT;
    protections_dPmaslo_gaz_less100_inCommand_ARM : UINT;
    protections_dPmaslo_gaz_less100_status : UDINT;
    protections_Reg_vozb_off_inCommand_ARM : UINT;
    protections_Reg_vozb_off_status : UDINT;
    protections_Fail_chastotnii_pusk_inCommand_ARM : UINT;
    protections_Fail_chastotnii_pusk_status : UDINT;
    protections_Off_avar_vikluchatel_inCommand_ARM : UINT;
    protections_Off_avar_vikluchatel_status : UDINT;
    protections_AOKC_SHKC_inCommand_ARM : UINT;
    protections_AOKC_SHKC_status : UDINT;
    protections_AO_PRU_inCommand_ARM : UINT;
    protections_AO_PRU_status : UDINT;
    protections_AO_ot_SHU_inCommand_ARM : UINT;
    protections_AO_ot_SHU_status : UDINT;
    protections_mvOff_inCommand_ARM : UINT;
    protections_mvOff_status : UDINT;
    protections_Kran1_sdvig_inCommand_ARM : UINT;
    protections_Kran1_sdvig_status : UDINT;
    protections_Kran2_sdvig_inCommand_ARM : UINT;
    protections_Kran2_sdvig_status : UDINT;
  END_VAR

  protections.Topornogo_podshipnika_EDT_1.inCommand_ARM := UINT_TO_WORD(protections_Topornogo_podshipnika_EDT_1_inCommand_ARM);

  protections.Toy_podshipnika_EDT_2.inCommand_ARM := UINT_TO_WORD(protections_Toy_podshipnika_EDT_2_inCommand_ARM);

  protections.Toy_podshipnika_kol_EDT_3.inCommand_ARM := UINT_TO_WORD(protections_Toy_podshipnika_kol_EDT_3_inCommand_ARM);

  protections.Toy_podshipnika_kol_EDT_4.inCommand_ARM := UINT_TO_WORD(protections_Toy_podshipnika_kol_EDT_4_inCommand_ARM);

  protections.To_podshipnika_shest_red_EDT_5.inCommand_ARM := UINT_TO_WORD(protections_To_podshipnika_shest_red_EDT_5_inCommand_ARM);

  protections.To_podshipnika_shest_red_EDT_6.inCommand_ARM := UINT_TO_WORD(protections_To_podshipnika_shest_red_EDT_6_inCommand_ARM);

  protections.To_podshipnika_N_EDT_7.inCommand_ARM := UINT_TO_WORD(protections_To_podshipnika_N_EDT_7_inCommand_ARM);

  protections.To_podshipnika_svob_konca_EDT_8.inCommand_ARM := UINT_TO_WORD(protections_To_podshipnika_svob_konca_EDT_8_inCommand_ARM);

  protections.Ty_podshipnika_rab_kol_EDT_9.inCommand_ARM := UINT_TO_WORD(protections_Ty_podshipnika_rab_kol_EDT_9_inCommand_ARM);

  protections.Typornogo_podshipnika_nerab_kolodok_HT_10.inCommand_ARM := UINT_TO_WORD(protections_Typornogo_podshipnika_nerab_kolodok_HT_10_inCommand_ARM);

  protections.Tgaza_na_vyhode_H.inCommand_ARM := UINT_TO_WORD(protections_Tgaza_na_vyhode_H_inCommand_ARM);

  protections.Os_sdvig_nagnetatelja_plus.inCommand_ARM := UINT_TO_WORD(protections_Os_sdvig_nagnetatelja_plus_inCommand_ARM);

  protections.Os_sdvig_nagnetatelja_minus.inCommand_ARM := UINT_TO_WORD(protections_Os_sdvig_nagnetatelja_minus_inCommand_ARM);

  protections.Pgaza_na_vyhode_nagnetatelia_GPA_STOP.inCommand_ARM := UINT_TO_WORD(protections_Pgaza_na_vyhode_nagnetatelia_GPA_STOP_inCommand_ARM);

  protections.Pgaza_na_vhode_nagnetatelia_GPA_STOP.inCommand_ARM := UINT_TO_WORD(protections_Pgaza_na_vhode_nagnetatelia_GPA_STOP_inCommand_ARM);

  protections.Pgaza_na_vyhode_nagnetatelia.inCommand_ARM := UINT_TO_WORD(protections_Pgaza_na_vyhode_nagnetatelia_inCommand_ARM);

  protections.dPmaslo_gaz.inCommand_ARM := UINT_TO_WORD(protections_dPmaslo_gaz_inCommand_ARM);

  protections.Pmaslo_sm_nizkoe.inCommand_ARM := UINT_TO_WORD(protections_Pmaslo_sm_nizkoe_inCommand_ARM);

  protections.Pmaslo_sm_vysokoe.inCommand_ARM := UINT_TO_WORD(protections_Pmaslo_sm_vysokoe_inCommand_ARM);

  protections.Vibro_skorost_OPED_T1.inCommand_ARM := UINT_TO_WORD(protections_Vibro_skorost_OPED_T1_inCommand_ARM);

  protections.Vibro_skorost_OPED_T2.inCommand_ARM := UINT_TO_WORD(protections_Vibro_skorost_OPED_T2_inCommand_ARM);

  protections.Vibro_skorost_OYP_kolesa_ED_T3.inCommand_ARM := UINT_TO_WORD(protections_Vibro_skorost_OYP_kolesa_ED_T3_inCommand_ARM);

  protections.Vibro_skorost_OP_kolesa_RH_T4.inCommand_ARM := UINT_TO_WORD(protections_Vibro_skorost_OP_kolesa_RH_T4_inCommand_ARM);

  protections.Vibro_skorost_OP_shesterni_RED_T5.inCommand_ARM := UINT_TO_WORD(protections_Vibro_skorost_OP_shesterni_RED_T5_inCommand_ARM);

  protections.Vibro_skorost_OP_shesterni_RED_T6.inCommand_ARM := UINT_TO_WORD(protections_Vibro_skorost_OP_shesterni_RED_T6_inCommand_ARM);

  protections.dPmaslo_gaz_less100.inCommand_ARM := UINT_TO_WORD(protections_dPmaslo_gaz_less100_inCommand_ARM);

  protections.Reg_vozb_off.inCommand_ARM := UINT_TO_WORD(protections_Reg_vozb_off_inCommand_ARM);

  protections.Fail_chastotnii_pusk.inCommand_ARM := UINT_TO_WORD(protections_Fail_chastotnii_pusk_inCommand_ARM);

  protections.Off_avar_vikluchatel.inCommand_ARM := UINT_TO_WORD(protections_Off_avar_vikluchatel_inCommand_ARM);

  protections.AOKC_SHKC.inCommand_ARM := UINT_TO_WORD(protections_AOKC_SHKC_inCommand_ARM);

  protections.AO_PRU.inCommand_ARM := UINT_TO_WORD(protections_AO_PRU_inCommand_ARM);

  protections.AO_ot_SHU.inCommand_ARM := UINT_TO_WORD(protections_AO_ot_SHU_inCommand_ARM);

  protections.mvOff.inCommand_ARM := UINT_TO_WORD(protections_mvOff_inCommand_ARM);

  protections.Kran1_sdvig.inCommand_ARM := UINT_TO_WORD(protections_Kran1_sdvig_inCommand_ARM);

  protections.Kran2_sdvig.inCommand_ARM := UINT_TO_WORD(protections_Kran2_sdvig_inCommand_ARM);
END_FUNCTION_BLOCK

FUNCTION_BLOCK OPC_IM_SET
  VAR_EXTERNAL
    Im : ImConfig;
    IM_Kran1_status : UDINT;
    IM_Kran1_inCommand_ARM : UINT;
    IM_Kran2_status : UDINT;
    IM_Kran2_inCommand_ARM : UINT;
    IM_Kran3_status : UDINT;
    IM_Kran3_inCommand_ARM : UINT;
    IM_Kran3b_status : UDINT;
    IM_Kran3b_inCommand_ARM : UINT;
    IM_Kran4_status : UDINT;
    IM_Kran4_inCommand_ARM : UINT;
    IM_Kran5_status : UDINT;
    IM_Kran5_inCommand_ARM : UINT;
    IM_Kran6_status : UDINT;
    IM_Kran6_inCommand_ARM : UINT;
    IM_nu1_status : UDINT;
    IM_nu1_inCommand_ARM : UINT;
    IM_nu2_status : UDINT;
    IM_nu2_inCommand_ARM : UINT;
    IM_pns_status : UDINT;
    IM_pns_inCommand_ARM : UINT;
    IM_v1_Avom_status : UDINT;
    IM_v1_Avom_inCommand_ARM : UINT;
    IM_v2_Avom_status : UDINT;
    IM_v2_Avom_inCommand_ARM : UINT;
    IM_v3_Avom_status : UDINT;
    IM_v3_Avom_inCommand_ARM : UINT;
    IM_v4_Avom_status : UDINT;
    IM_v4_Avom_inCommand_ARM : UINT;
    IM_mv_status : UDINT;
    IM_mv_inCommand_ARM : UINT;
    IM_KaloriferAVOM_status : UDINT;
    IM_KaloriferAVOM_inCommand_ARM : UINT;
    IM_CMN_status : UDINT;
    IM_CMN_inCommand_ARM : UINT;
    IM_TEN_kollectora_status : UDINT;
    IM_TEN_kollectora_inCommand_ARM : UINT;
    IM_TEN_MB_status : UDINT;
    IM_TEN_MB_inCommand_ARM : UINT;
    IM_SingleSignals_dP_maslo_gaz_Less100_status : UDINT;
    IM_SingleSignals_dp_kran1_Less100_status : UDINT;
    IM_SingleSignals_Razreshenie_zagruzki_dvig_status : UDINT;
    IM_SingleSignals_Vozbud_gotovnost_status : UDINT;
    IM_SingleSignals_Vozbud_neispr_tsepey_upr_AVR_pit_status : UDINT;
    IM_SingleSignals_Vozbud_neispravnost_status : UDINT;
    IM_SingleSignals_SHAVR1_v_rabote_status : UDINT;
    IM_SingleSignals_SHAVR2_v_rabote_status : UDINT;
    IM_SingleSignals_Avariinoe_otkluch_vikluchatelya_status : UDINT;
    IM_SingleSignals_Assinhronnii_hod_peregruzka_status : UDINT;
    IM_SingleSignals_SHU_v_GPA_vkluch_status : UDINT;
    IM_SingleSignals_SHP_v_GPA_vkluch_status : UDINT;
    IM_SingleSignals_QF1_on_status : UDINT;
    IM_SingleSignals_QF2_on_status : UDINT;
    IM_SingleSignals_QF23_on_status : UDINT;
    IM_SingleSignals_QF4_QF5_on_status : UDINT;
    IM_SingleSignals_QF6_QF7_on_status : UDINT;
    IM_SingleSignals_QF8_QF9_on_status : UDINT;
    IM_SingleSignals_QF10_QF11_on_status : UDINT;
    IM_SingleSignals_QF12_QF13_on_status : UDINT;
    IM_SingleSignals_QF14_QF15_on_status : UDINT;
    IM_SingleSignals_QF22_on_status : UDINT;
    IM_SingleSignals_NS_G1_G2_status : UDINT;
    IM_SingleSignals_NS_G3_G4_status : UDINT;
    IM_SingleSignals_NS_G15_G16_status : UDINT;
    IM_SingleSignals_NS_G17_status : UDINT;
    IM_SingleSignals_NS_G5_G6_status : UDINT;
    IM_SingleSignals_NS_G7_G8_status : UDINT;
    IM_SingleSignals_NS_G18_G19_status : UDINT;
    IM_SingleSignals_NS_G10_G11_status : UDINT;
    IM_SingleSignals_NS_G13_G14_status : UDINT;
    IM_SingleSignals_Uroven_masla_akkum_status : UDINT;
    IM_SingleSignals_NKU1_GPA_on_status : UDINT;
    IM_SingleSignals_NKU2_GPA_on_status : UDINT;
    IM_SingleSignals_AO_KC_ot_SHKS_status : UDINT;
    IM_SingleSignals_AO_GPA_ot_SHU_status : UDINT;
    IM_SingleSignals_BEAO_srabotal_status : UDINT;
    IM_SingleSignals_Chastotny_pusk_status : UDINT;
    IM_SingleSignals_Neuspesh_chastotny_pusk_status : UDINT;
    IM_SingleSignals_Rezhim_ruchnogo_regulirovaniya_status : UDINT;
    IM_SingleSignals_Osnovnoy_regul_off_status : UDINT;
    IM_SingleSignals_Voltage_sekcii_norm_status : UDINT;
    IM_SingleSignals_Reactorny_pusk_status : UDINT;
    IM_SingleSignals_NO_GPA_ot_SHU_status : UDINT;
    IM_SingleSignals_AO_GPA_ot_PRU_status : UDINT;
    IM_SingleSignals_Nalichie_BP1_status : UDINT;
    IM_SingleSignals_Nalichie_BP2_status : UDINT;
    IM_SingleSignals_Nalichie_BP3_status : UDINT;
    IM_SingleSignals_Nalichie_BP4_status : UDINT;
    IM_SingleSignals_Nalichie_BP5_status : UDINT;
    IM_SingleSignals_Nalichie_BP6_status : UDINT;
    IM_SingleSignals_Nalichie_BP7_BP8_status : UDINT;
    IM_SingleSignals_Nalichie_BP9_BP10_status : UDINT;
    IM_SingleSignals_Nalichie_cepei_upravlen_mv_status : UDINT;
    IM_SingleSignals_Nalichie_220BEAO_status : UDINT;
    IM_SingleSignals_Nalichie_per_220_na_vhode_status : UDINT;
    IM_SingleSignals_Nalichie_post_220_na_vhode_status : UDINT;
    IM_SingleSignals_Nalichie_BP11_status : UDINT;
    IM_SingleSignals_Nalichie_BP12_status : UDINT;
    IM_SingleSignals_Dver_SHU_pered_otkrita_status : UDINT;
    IM_SingleSignals_Dver_SHU_zad_otkrita_status : UDINT;
    IM_SingleSignals_EO_GPA_ot_knopki_SHU_status : UDINT;
    IM_SingleSignals_EO_EGPA_ot_PRY_status : UDINT;
    IM_SingleSignals_Synchroniz_rezhima_K1_status : UDINT;
    IM_SingleSignals_Potok_ms_posle_AVOM_status : UDINT;
  END_VAR
